IF STATE = BYTE#1 AND NOT FIFO.FULL THEN (* Anmelden *)
	(* nur eintragen wenn maximale anzahl nicht ueberschritten wurde *)
	tmp := BYTE_TO_INT(ID);
	IF FIFO.Y[tmp] < FIFO.MAX_ID THEN
		FIFO.Y[tmp] := USINT_TO_BYTE(BYTE_TO_USINT(FIFO.Y[tmp]) + USINT#1); (* IP_ID Zähler +1 *)
		tmp := FIFO.NW; (* geht bei mir leider nicht anders *)
		FIFO.X[tmp] := ID;
		IF FIFO.NW = FIFO.TOP THEN FIFO.NW := 1; ELSE FIFO.NW := FIFO.NW + 1; END_IF;
		FIFO.FULL := FIFO.NW = FIFO.NR;
		FIFO.EMPTY := FALSE;
		STATE := BYTE#2; (* weiterschalten auf "Warten auf Freigabe" *)
		(*####################  DEBUG-MESSAGE  ###################################*)
		(*IF _debug_enable THEN
			LOG_CL.NEW_MSG := 'FIFO: ADD ID:~1';
			LOG_CL.PRINTF[1]  := BYTE_TO_STRING(ID);
			LOG_MSG();
		END_IF;*)
		(*########################################################################*)

	END_IF;
END_IF;

IF STATE = BYTE#2 AND NOT FIFO.EMPTY THEN (* check current stack element *)
	tmp := FIFO.NR; (* geht bei mir leider nicht anders *)
	IF ID = FIFO.X[tmp] THEN
	STATE := BYTE#3; (* weiterschalten auf "Zugriffsfreigabe" *)
	END_IF;
END_IF;

IF STATE = BYTE#4 AND NOT FIFO.EMPTY THEN (* remove from stack *)
	tmp := FIFO.NR; (* geht bei mir leider nicht anders *)
	IF ID = FIFO.X[tmp] THEN
		tmp := BYTE_TO_INT(ID); (* geht bei mir leider nicht anders *)
		FIFO.Y[tmp] := USINT_TO_BYTE(BYTE_TO_USINT(FIFO.Y[tmp]) - USINT#1); (* ID Zähler -1 *)
		IF FIFO.NR = FIFO.TOP THEN FIFO.NR := 1; ELSE FIFO.NR := FIFO.NR + 1; END_IF;
		FIFO.EMPTY := FIFO.NR = FIFO.NW;
		FIFO.FULL := FALSE;
		(*####################  DEBUG-MESSAGE  ###################################*)
		(*IF _debug_enable THEN
			LOG_CL.NEW_MSG := 'FIFO: REMOVE ID:~1';
			LOG_CL.PRINTF[1]  := BYTE_TO_STRING(ID);
			LOG_MSG();
		END_IF;*)
		(*########################################################################*)
	END_IF;
	STATE := BYTE#5; (* "Remove done" *)
END_IF;

(* revision history
ks	18. oct. 2008	rev 1.0
	original version

*)

END_FUNCTION_BLOCK

// oscat_network/POUs/OTHER/ELEMENT_GET
FUNCTION ELEMENT_GET : STRING(ELEMENT_LENGTH)
VAR_INPUT
	SEP : BYTE;
	POS : INT;
END_VAR
VAR_IN_OUT
	ELEMENT : STRING(ELEMENT_LENGTH);
END_VAR
VAR
	i : INT := 1;
	o : INT := 1;
	pt : POINTER TO ARRAY[1..ELEMENT_LENGTH] OF BYTE;
	po : POINTER TO ARRAY[1..ELEMENT_LENGTH] OF BYTE;
	cnt: INT;
	c: BYTE;
END_VAR

(*
version 1.0	05. apr. 2011
programmer 	ks
tested by		kst

ELEMENT_GET liefert das element an der stelle pos einer liste.
die liste liegt als string von elementen vor die mit den zeichen SEP separiert sind.

*)

(* load pointers *)
pt := ADR(ELEMENT);
po := ADR(ELEMENT_GET);

(* search for the n-th occurence of a separation character and store position in i *)
WHILE (cnt < pos) AND (i < ELEMENT_LENGTH) AND (pt^[i] > 0) DO
	IF pt^[i] = sep THEN cnt := cnt + 1; END_IF;
	i := i + 1;
END_WHILE;

(* copy the list element to output *)
IF i < ELEMENT_LENGTH THEN c := pt^[i]; END_IF;
WHILE (c <> sep) AND (c > 0) AND (o < ELEMENT_LENGTH) AND (i < ELEMENT_LENGTH) DO
	po^[o] :=pt^[i];
	o := o + 1;
	i := i + 1;
	c := pt^[i];
END_WHILE;

(* terminate the output string *)
po^[o] := 0;

(* revision histroy
ks 05. apr. 2011	rev 1.0
	original release

*)

END_FUNCTION

// oscat_network/POUs/OTHER/ELEMENT_COUNT
FUNCTION ELEMENT_COUNT : INT
VAR_INPUT
	SEP : BYTE;
END_VAR
VAR_IN_OUT
	ELEMENT : STRING(ELEMENT_LENGTH);
END_VAR
VAR
	pt : POINTER TO ARRAY[1..ELEMENT_LENGTH] OF BYTE;
	l: INT;
	pos: INT;
END_VAR

(*
version 1.0	05. apr. 2011
programmer 	hugo
tested by		oscat

ELEMENT_COUNT liefert die anzahl der elemente einer liste.
die liste liegt als string von elementen vor die mit den zeichen SEP separiert sind.

*)

IF ELEMENT = '' THEN
	ELEMENT_COUNT := 0;
ELSE
	PT := ADR(ELEMENT);
	ELEMENT_COUNT := 1;
	l := LEN(ELEMENT);
	FOR pos := 1 TO l DO
		IF pt^[pos] = SEP THEN ELEMENT_COUNT := ELEMENT_COUNT + 1; END_IF;
	END_FOR;
END_IF;

(* revision histroy
ks	5. apr. 2011	rev 1.0
	original release

*)

END_FUNCTION

// oscat_network/POUs/DATA_LOG/DLOG_FILE_TO_SMTP_1
(* @OBJECTFLAGS := '0, 8' *)
FUNCTION_BLOCK DLOG_FILE_TO_SMTP_1
VAR_IN_OUT
	SERVER : STRING;
	MAILFROM : STRING;
	MAILTO : STRING(STRING_LENGTH);
	SUBJECT : STRING;
	BODY : STRING(STRING_LENGTH);
	X : DLOG_DATA;
END_VAR
VAR_INPUT
	FILE_DELETE : BOOL;
	TIMEOUT : TIME := T#30s;
	DTI : DT;
	DTI_OFFSET : INT;
	RETRY : INT;
	RETRY_TIME : TIME := T#30s;
	DNS_IP4 : DWORD;
END_VAR
VAR_OUTPUT
	DONE : BOOL;
	BUSY : BOOL;
	ERROR_C : DWORD;
	ERROR_T : BYTE;
END_VAR
VAR
	UCBD : UNI_CIRCULAR_BUFFER_DATA;
	UCB : UNI_CIRCULAR_BUFFER;
	SMTP_CLIENT : SMTP_CLIENT;
	WT_1 : TON;
	ftrig_old : BOOL;
	files : STRING(STRING_LENGTH);
	step : INT;
	smtp_busy : BOOL;
	smtp_done : BOOL;
	cnt : INT;

	(*LOG_MSG : LOG_MSG;
	_debug_enable : BOOL := TRUE;*)
END_VAR

(*
version 1.2		26. july. 2011
programmer		ks
tested by			ks

DLOG_FILE_TO_SMTP der Baustein versendet die vom DLOG_STORE_FILE_CSV erzeugten Dateien als Email
*)

(* neue Filenamen speichern *)
IF X.NEW_FILE_RTRIG AND ftrig_old = FALSE THEN
	UCBD.D_HEAD := 1;
	UCBD.D_MODE := 1;
	UCBD.D_STRING := X.NEW_FILE;
	UCB(DATA:=UCBD); (* Daten eintragen *)
END_IF;
ftrig_old := X.NEW_FILE_RTRIG;

CASE step OF

00:	IF UCBD.BUF_COUNT > 0 AND smtp_busy = FALSE THEN
		UCBD.D_MODE := 12; (* Daten lesen und löschen *)
		UCB(DATA:=UCBD);
		files := UCBD.D_STRING;
		IF FILE_DELETE THEN
			files := CONCAT(files,';#DEL#');
		END_IF;
		cnt := 0;
		step := 10;
	END_IF;

10:	IF smtp_busy = FALSE THEN
		IF smtp_done THEN
			(*####################  DEBUG-MESSAGE  ###################################*)
			(*IF _debug_enable THEN
				LOG_CL.NEW_MSG := 'F_T_SMTP: /FILE OK >~1<';
				LOG_CL.PRINTF[1] := files;
				LOG_MSG();
			END_IF;*)
			(*########################################################################*)
			step := 0;
		ELSE
			step := 20; (* pause nach error *)
		END_IF;
	END_IF;

20:	IF WT_1.Q THEN (* Wartezeit *)
		cnt := cnt - 1;
		IF RETRY = 0 THEN (* Transfer unbegrenzt wiederholen *)
			(*####################  DEBUG-MESSAGE  ###################################*)
			(*IF _debug_enable THEN
				LOG_CL.NEW_MSG := 'F_T_SMTP: Auftrag unbegrenzt wiederholen /file: ~2';
				LOG_CL.PRINTF[2] := files;
				LOG_MSG();
			END_IF;*)
			(*########################################################################*)
			step := 10; (* Transfer wiederholen *)
		ELSIF cnt >= 0 THEN
			(*####################  DEBUG-MESSAGE  ###################################*)
			(*IF _debug_enable THEN
				LOG_CL.NEW_MSG := 'F_T_SMTP: Auftrag wiederholen /cnt: ~1 /file: ~2';
				LOG_CL.PRINTF[1] := INT_TO_STRING(cnt);
				LOG_CL.PRINTF[2] := files;
				LOG_MSG();
			END_IF;*)
			(*########################################################################*)
			step := 10; (* Transfer wiederholen *)
		ELSE
			(*####################  DEBUG-MESSAGE  ###################################*)
			(*IF _debug_enable THEN
				LOG_CL.NEW_MSG := 'F_T_SMTP: Auftrag verworfen /file: ~2';
				LOG_CL.PRINTF[2] := files;
				LOG_MSG();
			END_IF;*)
			(*########################################################################*)
			step := 0; (* Auftrag verwerfen *)
		END_IF;
	END_IF;

END_CASE;

BUSY := step = 10;
DONE := step = 0;
WT_1(IN:= step = 20, PT:= RETRY_TIME);

SMTP_CLIENT(
	ACTIVATE:= BUSY,
	TIMEOUT:= TIMEOUT,
	DTI:= DTI,
	DTI_OFFSET:= DTI_OFFSET,
	DNS_IP4:= DNS_IP4,
	SERVER:= SERVER,
	MAILFROM:= MAILFROM,
	MAILTO:= MAILTO,
	SUBJECT:= SUBJECT,
	BODY:= BODY,
	FILES:= FILES,
	DONE=> smtp_done,
	BUSY=> smtp_busy,
	ERROR_C=> ERROR_C,
	ERROR_T=> ERROR_T
	);

(* revision history

ks	01. jan. 2011	rev 1.0
	original version

ks	28. apr. 2011	rev 1.1
	stringfehler bei option 'file_delete'

ks	26. july. 2011	rev 1.2
	Codeoptimierung D_MODE 12
*)

END_FUNCTION_BLOCK

// oscat_network/POUs/NETWORK/SMTP_CLIENT
FUNCTION_BLOCK SMTP_CLIENT
VAR_INPUT
	ACTIVATE : BOOL;
	TIMEOUT : TIME;
	DTI : DT;
	DTI_OFFSET : INT;
	DNS_IP4 : DWORD;
END_VAR
VAR_OUTPUT
	DONE : BOOL;
	BUSY : BOOL;
	ERROR_C : DWORD;
	ERROR_T : BYTE;
END_VAR
VAR_IN_OUT
	SERVER : STRING;
	MAILFROM : STRING;
	MAILTO : STRING(STRING_LENGTH);
	SUBJECT : STRING;
	BODY : STRING(STRING_LENGTH);
	FILES : STRING(STRING_LENGTH);
END_VAR
VAR
	IP_C : IP_C; (* IP_Control Verwaltungsstruktur *)
	S_BUF : NETWORK_BUFFER;
	R_BUF : NETWORK_BUFFER;
	F_BUF : NETWORK_BUFFER;
	URL_DATA : url;
	DNS_CLIENT : DNS_CLIENT;
	IPC : IP_CONTROL;
	FS : FILE_SERVER;
	FSD : FILE_SERVER_DATA;
	BASE64_ENCODE_STR : BASE64_ENCODE_STR;
	BASE64_ENCODE_STREAM : BASE64_ENCODE_STREAM;
	fpd : FILE_PATH_DATA;
	MD5_CRAM_AUTH : MD5_CRAM_AUTH;
	MD5_RUN : BOOL;
	activate_last : BOOL;
	step : INT;
	snd_step : INT;
	str1 : STRING(STRING_LENGTH);
	str2 : STRING(STRING_LENGTH);
	str3 : STRING;
	snd_text :	STRING(STRING_LENGTH);
	snd_lf_cnt : INT;
	rcv_text :	STRING(STRING_LENGTH);
	rcv_s : STRING(3);
	rcv_state : INT;
	auth_names : STRING := ' PLAIN; LOGIN; CRAM-MD5';
	auth_state : BYTE;
	TON_WAIT : TON;
	last_step : INT;
	next_step : INT;
	timeout2 : TIME;
	timeout3 : TIME;
	last_block : BOOL;
	file_delete : BOOL;
	esmtp : BOOL;
	cnt1 : INT;
	cnt2 : INT;
	cnt3 : INT;
	cnt4 : INT;
	idx1 : INT;
	idx2 : INT;
	idx3 : INT;
	snd_idx : INT;
	snd_enable : BOOL;
	i1 : INT;
	b64_done : BOOL;
	b64_start : BOOL;
	b64_max : UINT := 2880; (* short = 960 / long = 2880 *)
	b64_buf1 : ARRAY [0..47] OF BYTE;
	b64_buf2 : ARRAY [0..63] OF BYTE;
	b64_size1 : INT;
	b64_size2 : INT;
	b64_lf : BOOL;
	b64_str1	: STRING(144);
	b64_str2	: STRING(192);
	md5_user : STRING(64);
	md5_password : STRING(64);
	md5_b64_ts : STRING(64);
	md5_auth_key : STRING(192);
	ip_c_red_disable : BOOL; (* IP_CONTROL - Remote Disconnect Error unterdrücken *)

	(*LOG_MSG : LOG_MSG;
	_debug_enable : BOOL := TRUE;*)
END_VAR

(*
version 1.3		30. may 2011
programmer		ks
tested by			ks

SMTP_CLIENT versendet Email an verschiedene Emailadressen mit optionalen Dateianhängen.



mögliche Rückgabecodes:

Grad der Schwere
 
Die erste Stelle des Rückgabecodes gibt den Grad der Schwere an:
1yz Vorläufige positive Antwort
2yz Antwort über positiven Abschluss 
3yz Positive Zwischenantwort 
4yz Antwort über vorübergehenden negativen Abschluss 
5yz Permanente negative Antwort 
 
Die zweite Stelle gibt die Kategorie der Antwort an: 
x0z Syntaxfehler 
x1z Information 
x2z Verbindung 
x3z Nicht festgelegt 
x4z Nicht festgelegt 
x5z Mail-System 
 
Die dritte Stelle dient zur genaueren Bestimmung der Kategorie. 

Betriebsprotokolle enthalten folgende Codes: 
211 	Systemstatus oder Hilfe-Antwort des Systems  
214 	Hilfe-Nachricht - Informationen zur Verwendung des Empfängers oder zur  
      	Bedeutung eines bestimmten nicht standardmäßigen Befehls; wobei  
      	diese Antwort nur für Personen hilfreich ist, nicht für Systeme 
220 	Service ready (Dienst bereit) 
221 	Service closing transmission channel (Dienst schließt Übertragungskanal) 
235  Authentication succeeded (Authentifizierung erfolgreich)
250 	Requested mail action okay, completed (angeforderte Mail-Maßnahme ok und abgeschlossen) 
251 	User not local; will forward to (Benutzer nicht lokal; Weiterleitung an) 
252 	Cannot VRFY user, but will accept message and attempt delivery (kann Benutzer nicht überprüfen, aber akzeptiert Nachricht und versucht Auslieferung) 
354 	Start mail input; end with. (Mail-Eingabe starten; Ende mit .) 
421 	Service not available, closing transmission channel 	(Dienst nicht verfügbar, Übertragungskanal wird geschlossen) diese Antwort kann auf jeden Befehl folgen, wenn der Dienst weiß, dass er beendet werden muss 
450 	Requested mail action not taken: mailbox unavailable (angeforderte E-Mail-Maßnahme nicht ausgeführt, Mailbox nicht  verfügbar) - z. B. weil Mailbox besetzt 
451	 Requested action aborted: local error in processing (angeforderte Maßnahme abgebrochen: lokaler Fehler bei der Verarbeitung) 
452 	Requested action not taken: insufficient system storage (angeforderte Maßnahme abgebrochen: Systemspeicher nicht ausreichend) 
500 	Syntax error, command unrecognized (Syntaxfehler, Befehl nicht erkannt) - z. B. weil Befehlszeile zu lang 
501 	Syntax error in parameters or arguments (Syntaxfehler in Parametern oder Argumenten) 
502 	Command not implemented (Befehl nicht implementiert) 
504 	Command parameter not implemented (Befehlsparameter nicht implementiert) 
550 	Requested action not taken: mailbox unavailable (Angeforderte Maßnahme nicht ausgeführt: Mailbox nicht verfügbar) 
551 	User not local; please try (Benutzer nicht lokal; versuchen Sie es mit) 
552 	Requested mail action aborted: exceeded storage allocation (angeforderte Mail-Maßnahme abgebrochen: Speicherplatzzuweisung überschritten) 
553 	Requested action not taken: mailbox name not allowed (angeforderte Maßnahme nicht ausgeführt: Mailboxname nicht zulässig) 
554 	Transaction failed (Transaktion fehlgeschlagen) 

#########################
ERROR_T

1 = DNS_CLIENT
2 = SMTP Steuerkanal
4 = FILE_SERVER
5 = Ablaufstörung
#########################

*)

CASE step OF

00:	IF ACTIVATE AND NOT activate_last THEN
		TIMEOUT := MAX(T#10s,TIMEOUT);
		timeout2 := TIMEOUT + T#1s;
		timeout3 := TIMEOUT / 2;
		DONE := FALSE;
		ip_c_red_disable := FALSE;
		ERROR_C := DWORD#0;
		ERROR_T := BYTE#0;
		FSD.ERROR := BYTE#0;
		file_delete := FALSE;
		URL_DATA := STRING_TO_URL(STR:=SERVER,DEFAULT_PROTOCOL:='',DEFAULT_PATH:='/');
		idx1 := FIND(URL_DATA.USER,'%'); (* % Zeichen auf @ ändern *)
		IF idx1 > 0 THEN
			URL_DATA.USER := REPLACE(URL_DATA.USER,'@',1,idx1);
		END_IF;
		esmtp := LEN(URL_DATA.PASSWORD) > 0; (* SMTP oder ExtendedSMTP *)
		step := 10;
	END_IF;

10:	IF DNS_CLIENT.DONE THEN
		step := 20;
	ELSIF DNS_CLIENT.ERROR <> DWORD#0 THEN
		ERROR_C := DNS_CLIENT.ERROR;
		ERROR_T := BYTE#1;
		step := 980;
	END_IF;

20:	(* SMTP Kommunikation einrichten *)
	IP_C.C_PORT := SEL(URL_DATA.PORT = WORD#0,URL_DATA.PORT,WORD#25); (* Portnummer eintragen *)
  	IP_C.C_IP := DNS_CLIENT.IP4; (* IP eintragen *)
  	IP_C.C_MODE := BYTE#0; (* Mode: TCP+ACTIV+PORT *)
  	IP_C.TIME_RESET := TRUE; (* Zeitueberwachung rücksetzen *)
  	IP_C.C_ENABLE := TRUE; (* Verbindungsaufbau freigeben *)
  	IP_C.R_OBSERVE := TRUE; (* Empfangsueberwachung *)
	R_BUF.SIZE := UINT#0;
	snd_enable := TRUE; (* sofortiges senden erlauben *)
	snd_idx := 0;
	step := 30;

30:	IF rcv_state = 220 THEN (* 220 = Service ready *)
		IF esmtp THEN
			snd_text := 'EHLO OSCAT'; (* ExtendedSMTP *)
			next_step := 40;
		ELSE
			snd_text := 'HELO OSCAT'; (* SMTP *)
			next_step := 90;
		END_IF;
		snd_lf_cnt := 1;
	END_IF;

40:	IF rcv_state = 250 THEN (* 250 = Requested mail action okay, completed  *)
		auth_state := BYTE#0;
		str1 := auth_names;
		idx1 := 0;
		idx2 := 1900;
		step := 50;
	END_IF;

50:	str2 := ELEMENT_GET(59, idx1, str1); (* Trennzeichen >;< *)
	IF LEN(str2) > 0 THEN
		IF FIND(rcv_text,str2) > 0 THEN
			auth_state := BIT_LOAD_B(auth_state, TRUE, idx1);
			str3 := str2; (* aktuellen AUTH-Type Namen sichern *)
			idx2 := 1000 + (idx1 * 100); (* Schritt berechnen *)
		END_IF;
		idx1 := idx1 + 1;
	ELSE
		step := 60;
	END_IF;

60:	IF rcv_state = 250 THEN (* 250 = Requested mail action okay, completed  *)
		snd_text := CONCAT('AUTH',str3);
		next_step := idx2; (* mit den jeweiligen Authentifizierung Schritten fortfahren *)
	END_IF;

 (* ++++++++++++++++++++++++++++++++++++++++++++++++++++++*)

90:	IF rcv_state = 235 OR rcv_state = 250 THEN (* 235 = Authentication successful / 250 Requested mail action okay *)
		str2 := MAILFROM;
		str1 := ELEMENT_GET(59, 1, str2);(* Angezeigter Name lesen , Trennzeichen >;< *)
		IF LEN(str1) > 0 THEN
			str3 := INSERT('"" ', str1, 1);
		ELSE
			str3 := '';
		END_IF;
		str1 := ELEMENT_GET(59, 0, str2);(* MAILFROM lesen , Trennzeichen >;< *)
		str2 := INSERT('MAIL FROM: <>', str1, 12);
		snd_text := INSERT(str2, str3, 11);
		str3 := snd_text; (* zur wiederverwendung speichern *)
		next_step := 95;
		cnt1 := ELEMENT_COUNT(35, MAILTO); (* Trennzeichen >#< , Anzahl der Blöcke bestimmen *)
		cnt2 := 0;
	END_IF;

95:	IF rcv_state = 250 THEN (* 250 = Requested mail action okay *)
		IF cnt2 < cnt1 THEN
			str1 := ELEMENT_GET(35, cnt2, MAILTO);(* Trennzeichen >#< *)
			cnt3 := ELEMENT_COUNT(59, str1); (* Trennzeichen >;< , Anzahl der Sub-Blöcke bestimmen *)
			cnt4 := 0;
			cnt2 := cnt2 + 1;
			step := 100; (* Blockinhalt auswerten *)
		ELSE
			step := 110; (* alle Blöcke bearbeitet *)
		END_IF;
	END_IF;

100:	IF rcv_state = 250 THEN (* 250 = Requested mail action okay *)
		IF cnt4 < cnt3 THEN
			str2 := ELEMENT_GET(59, cnt4, str1); (* Trennzeichen >;< *)
			snd_text := INSERT('RCPT TO: <>', str2, 10);
			cnt4 := cnt4 + 1;
			next_step := 100;
		ELSE
			step := 95;
		END_IF;
	END_IF;

110:	IF rcv_state = 250 THEN (* 250 = Requested mail action okay *)
		snd_text := 'DATA';
		next_step := 120;
	END_IF;

120:	IF rcv_state = 354 THEN (* 354 = Start mail input; end with. *)
		snd_enable := FALSE;
		snd_text := REPLACE(str3, 'From', 9, 1); (* 'MAIL FROM' durch "From" ersetzen *)
		cnt2 := 0;
		cnt1 := MIN(2,cnt1); (* BlindCopy Block ausblenden *)
		step := 200;
	END_IF;

200:	IF snd_step = 0 THEN
		IF cnt2 < cnt1 THEN
			str1 := ELEMENT_GET(35, cnt2, MAILTO);(* Trennzeichen >#< *)
			cnt3 := ELEMENT_COUNT(59, str1); (* Trennzeichen >;< , Anzahl der Sub-Blöcke bestimmen *)
			cnt4 := 0;
			cnt2 := cnt2 + 1;
			str3 := SEL(cnt2 = 1,'Cc: <>','To: <>');
			step := 205; (* Blockinhalt auswerten *)
		ELSE
			step := 210; (* alle Blöcke bearbeitet *)
		END_IF;
	END_IF;

205:	IF snd_step = 0 THEN
		IF cnt4 < cnt3 THEN
			str2 := ELEMENT_GET(59, cnt4, str1); (* Trennzeichen >;< *)
			snd_text := INSERT(str3, str2, 5);
			cnt4 := cnt4 + 1;
		ELSE
			step := 200;
		END_IF;
	END_IF;

210:	IF snd_step = 0 THEN
		snd_text := CONCAT('Subject: ',SUBJECT);
		step := 220;
	END_IF;

220:	IF snd_step = 0 THEN
		DTI := UDINT_TO_DT(DT_TO_UDINT(DTI) + INT_TO_UDINT(- DTI_OFFSET * 60)); (* Minuten-Offset auf Sekunden umrechnen und addieren *)
		IF esmtp THEN (* ESMTP Format >Date: Thu, 21 May 1998 05:33:29 -0700< *)
			str2 := ';Mon;Tue;Wed;Thu;Fri;Sat;Sun';
			str1 := ELEMENT_GET(59, DAY_OF_WEEK(DT_TO_DATE(DTI)), str2);
			snd_text := CONCAT('Date: ',str1);
			str1 := DT_TO_STRF(DTI, 0, ', #H #E #A #N:#R:#T +0000', 1);
			snd_text := CONCAT(snd_text,str1);
		ELSE (* SMTP Format >Date: 21 May 98 05:33:29< *)
			snd_text := DT_TO_STRF(DTI, 0, 'Date: #G #E #B #N:#R:#T', 1);
		END_IF;
		step := 230;
	END_IF;

230:	IF snd_step = 0 THEN
		snd_text := 'MIME-Version: 1.0';
		step := 250;
	END_IF;

250:	IF snd_step = 0 THEN
		snd_text := 'Content-Type: multipart/mixed;boundary="x"';
		snd_lf_cnt := 2;
		step := 260;
	END_IF;

260:	IF snd_step = 0 THEN
		snd_enable := TRUE;
		snd_text := 'This is a multi-part message in MIME format.';
		step := 270;
	END_IF;

270:	IF snd_step = 0 THEN
		snd_enable := FALSE;
		snd_text := '--x';
		snd_lf_cnt := 1;
		step := 280;
	END_IF;

280:	IF snd_step = 0 THEN
		snd_text := 'Content-Type: text/plain; format=flowed; charset="iso-8859-1";';
		snd_text := CONCAT(snd_text,' reply-type=original'); (* PCWORX kann nur konstanten mit max 80 zeichen *)
		step := 290;
	END_IF;

290:	IF snd_step = 0 THEN
		snd_text := 'Content-Transfer-Encoding: 8bit';
		snd_lf_cnt := 2;
		step := 300;
	END_IF;

300:	IF snd_step = 0 THEN
		snd_enable := TRUE;
		snd_text := BODY;
		snd_lf_cnt := 2;
		step := 310;
	END_IF;

310:	IF snd_step = 0 THEN
		cnt1 := ELEMENT_COUNT(59, FILES) - 1; (* Anzahl der Dateien *)
		step := 400;
	END_IF;

(* +++++++++++++ File-Attachment ++++++++++++ *)
400:	IF cnt1 >= 0 THEN
		str1 := ELEMENT_GET(59, cnt1, FILES);
		FILE_PATH_SPLIT(FILENAME:=str1,X:=fpd); (* Datei-Path zerlegen *)
		IF fpd.FILENAME = '#DEL#' THEN
			file_delete := TRUE;
		ELSE
			step := 410;
		END_IF;
		cnt1 := cnt1 - 1;
	ELSE
		step := 800;
	END_IF;

410:	IF snd_step = 0 THEN
		snd_enable := FALSE;
		snd_text := '--x';
		snd_lf_cnt := 1;
		step := 420;
	END_IF;

420:	IF snd_step = 0 THEN
		snd_text := 'Content-Transfer-Encoding: BASE64';
		str2 := CONCAT(fpd.FILENAME,'"');
		step := 430;
	END_IF;

430:	IF snd_step = 0 THEN
		snd_text := CONCAT('Content-Type: application/octet-stream; name="',str2);
		step := 440;
	END_IF;

440:	IF snd_step = 0 THEN
		snd_enable := TRUE;
		snd_text := CONCAT('Content-Disposition: attachment; filename="',str2);
		snd_lf_cnt := 2;
		step := 450;
	END_IF;

450:	IF snd_step = 0 THEN
		FSD.FILENAME := str1; (* Dateiname *)
		FSD.OFFSET := UDINT#0; (* Start bei Dateianfang *)
		FSD.AUTO_CLOSE := T#0s; (* kein Auto-Close verwenden *)
		step := 460;
	END_IF;

460:	FSD.MODE := BYTE#1; (* vorhandene Datei zum lesen öffnen *)
	F_BUF.SIZE := b64_max; (* maximale länge einlesen *)
	idx1 := 0;
	idx2 := 0;
	step := 470;

470:	IF FSD.MODE = BYTE#0 AND FSD.ERROR = BYTE#0 THEN
		last_block := FSD.FILE_SIZE = FSD.OFFSET;
		b64_size1 := MIN(48,UINT_TO_INT(F_BUF.SIZE) - idx1);
		IF b64_size1 > 0 THEN
			idx3 := b64_size1 - 1;
			FOR i1 := 0 TO idx3 DO (* daten in BASE64 buffer kopieren *)
				b64_buf1[i1] := F_BUF.BUFFER[idx1];
				idx1 := idx1 + 1;
			END_FOR;
			BASE64_ENCODE_STREAM( SIZE1:= b64_size1, BUF1:= b64_buf1, BUF2:= b64_buf2, SIZE2=> b64_size2); (* BASE64 Kodierung *)
			idx3 := b64_size2 - 1;
			FOR i1 := 0 TO idx3 DO (* Daten aus BASE64 buffer kopieren *)
				S_BUF.BUFFER[idx2] := b64_buf2[i1];
				idx2 := idx2 + 1;
			END_FOR;
			b64_lf := TRUE;
			(*####################  DEBUG-MESSAGE  ###################################*)
			(*IF _debug_enable THEN
				LOG_CL.NEW_MSG := 'B64: FILE ~1 /SIZE ~2 /OFF ~3 /BSIZE ~4 /idx1 ~5 /idx2 ~6';
				LOG_CL.PRINTF[1] := FSD.FILENAME;
				LOG_CL.PRINTF[2] := UDINT_TO_STRING(FSD.FILE_SIZE);
				LOG_CL.PRINTF[3] := UDINT_TO_STRING(FSD.OFFSET);
				LOG_CL.PRINTF[4] := INT_TO_STRING(b64_size1);
				LOG_CL.PRINTF[5] := INT_TO_STRING(idx1);
				LOG_CL.PRINTF[6] := INT_TO_STRING(idx2);
				LOG_MSG();
			END_IF;*)
			(*########################################################################*)
		ELSE
			b64_lf := last_block;
			step := 480; (* block beendet  *)
		END_IF;
		IF b64_lf THEN
			S_BUF.BUFFER[idx2] := BYTE#16#0D;
			idx2 := idx2 + 1;
			S_BUF.BUFFER[idx2] := BYTE#16#0A;
			idx2 := idx2 + 1;
		END_IF;
		(*####################  DEBUG-MESSAGE  ###################################*)
		(*IF _debug_enable THEN
			LOG_CL.NEW_MSG := 'B64: exit ~1 /SIZE ~2 /OFF ~3 /eof ~4 /lf_cnt ~5';
			LOG_CL.PRINTF[1] := FSD.FILENAME;
			LOG_CL.PRINTF[2] := UDINT_TO_STRING(FSD.FILE_SIZE);
			LOG_CL.PRINTF[3] := UDINT_TO_STRING(FSD.OFFSET);
			LOG_CL.PRINTF[4] := BOOL_TO_STRING(last_block);
			LOG_CL.PRINTF[5] := INT_TO_STRING(snd_lf_cnt);
			LOG_MSG();
		END_IF;*)
		(*########################################################################*)
	END_IF;

480:	S_BUF.SIZE := INT_TO_UINT(idx2); (* Daten senden *)
	(*####################  DEBUG-MESSAGE  ###################################*)
	(*IF _debug_enable THEN
		LOG_CL.NEW_MSG := 'B64: tcp_send ~1';
		LOG_CL.PRINTF[1] := INT_TO_STRING(idx2);
		LOG_MSG();
	END_IF;*)
	(*########################################################################*)
	step := 490;

490:	IF S_BUF.SIZE = UINT#0 THEN (* warten bis alle daten gesendet sind *)
		step := SEL(last_block ,460,400);
	END_IF;

(* ++++++++++++++++++++++++++++++++++++++++ *)

800:	IF snd_step = 0 THEN
		snd_enable := FALSE;
		snd_text := '--x--';
		snd_lf_cnt := 2;
		step := 810;
	END_IF;

810:	IF snd_step = 0 THEN
		snd_enable := TRUE;
		snd_text := '.';
		snd_lf_cnt := 1;
		step := 820;
	END_IF;

820:	IF rcv_state = 250 THEN (* 250 = Requested mail action okay *)
		snd_text := 'QUIT';
		ip_c_red_disable := TRUE;
		next_step := 830;
	END_IF;

830:	IF rcv_state = 221  OR TON_WAIT.ET > timeout3 THEN (* 221 = Service closing transmission channel *)
		step := 900;
	END_IF;

(* ================================================== *)

900:IF FILE_DELETE THEN (* Dateien nach transfer löschen *)
		cnt1 := ELEMENT_COUNT(59, FILES) - 1; (* Anzahl der Dateien *)
		step := 910;
	ELSE
		step := 950;
	END_IF;

910:	IF FSD.MODE = BYTE#0 AND FSD.ERROR = BYTE#0 THEN
		IF cnt1 >= 0 THEN
			str1 := ELEMENT_GET(59, cnt1, FILES);
			IF str1 <> '#DEL#' THEN
				FSD.FILENAME := str1;
				FSD.MODE := BYTE#4; (* File Remove *)
			END_IF;
			cnt1 := cnt1 - 1;
		ELSE
			step := 950;
		END_IF;
	END_IF;

950:DONE := TRUE;
	step := 980;

980:IP_C.C_ENABLE := FALSE; (* SMTP Steuerkanal schliessen *)
	S_BUF.SIZE := UINT#0;
	R_BUF.SIZE := UINT#0;
	snd_step := 0;
	next_step := 0;
	FSD.MODE := BYTE#5; (* Datei schliessen *)
	step := 990;

990:IF IP_C.C_STATE = BYTE#0 AND FSD.FILE_OPEN = FALSE THEN
		step := 0;
	END_IF;

(*  +++++++++++++++++ Authentifizierung +++++++++++++++++ *)

(* PLAIN ++++++++++++++++++++++++++++++++++++++++++++++++++++++++++ *)
1000:IF rcv_state = 334 THEN (* 334 = Authentifizierung  *)
		cnt1 := LEN(URL_DATA.USER);
		cnt2 := LEN(URL_DATA.PASSWORD);
		IF cnt1 + cnt2 <= 46 THEN (* USER + PASSWORD dürfen zusammen maximal 46 Zeichen haben *)
			b64_buf1[0] := BYTE#0;
			FOR i1 := 1 TO cnt1 DO
				b64_buf1[i1] := CODE(URL_DATA.USER, i1);
			END_FOR;
			b64_size1 := cnt1 + 1;
			b64_buf1[b64_size1] := BYTE#0;
			b64_size1 := b64_size1 + 1;
			FOR i1 := 1 TO cnt2 DO
				b64_buf1[b64_size1] := CODE(URL_DATA.PASSWORD, i1);
				b64_size1 := b64_size1 + 1;
			END_FOR;
			BASE64_ENCODE_STREAM( SIZE1:= b64_size1, BUF1:= b64_buf1, BUF2:= b64_buf2, SIZE2=> b64_size2); (* BASE64 Kodierung *)
			idx1 := b64_size2 - 1;
			FOR i1 := 0 TO idx1 DO
				S_BUF.BUFFER[i1] := b64_buf2[i1];
			END_FOR;
			S_BUF.BUFFER[b64_size2] := BYTE#16#0D;
			b64_size2 := b64_size2 + 1;
			S_BUF.BUFFER[b64_size2] := BYTE#16#0A;
			b64_size2 := b64_size2 + 1;
			S_BUF.SIZE := INT_TO_UINT(b64_size2);
			rcv_state := 0;
		END_IF;
		step := 90;
	END_IF;

(* LOGIN ++++++++++++++++++++++++++++++++++++++++++++++++++++++++++ *)
1100:IF rcv_state = 334 THEN (* 334 = Authentifizierung  *)
		b64_str1 := URL_DATA.USER;
		b64_start := TRUE; (* BASE64 kodierung von Username *)
		step := 1120;
	END_IF;

1120:IF b64_start AND b64_done THEN
		b64_start := FALSE;
		snd_text := b64_str2;
		next_step := 1130;
	END_IF;

1130:IF rcv_state = 334 THEN (* 334 = Password:  *)
		b64_str1 := URL_DATA.PASSWORD;
		b64_start := TRUE; (* BASE64 kodierung von Password *)
		step := 1140;
	END_IF;

1140:IF b64_start AND b64_done THEN
		b64_start := FALSE;
		snd_text := b64_str2;
		next_step := 90;
	END_IF;

(* CRAM-MD5 (Challenge-Response Authentication Mechanism, Message Digest 5) Authentifizierung auf Basis von MD5-HMAC-Algorithmus. *)
1200:IF rcv_state = 334 THEN (* 334 = Authentifizierung  *)
		md5_b64_ts := RIGHT(rcv_text,LEN(rcv_text) - 4);
		md5_user := URL_DATA.USER;
		md5_password := URL_DATA.PASSWORD;
		MD5_RUN := TRUE;
		step := 1220;
	END_IF;

1220:MD5_CRAM_AUTH(RUN:=MD5_RUN,USERNAME:=md5_user,PASSWORD:=md5_password,B64_TS:=md5_b64_ts,AUTH_KEY:=md5_auth_key);
	IF NOT MD5_RUN THEN
		snd_text := md5_auth_key;
		step := 90;
	END_IF;

(* keine Authentifizierung gefunden +++++++++++++++++++++++++++++++ *)
1900: ; (* Auf Laufzeitfehler warten *)

END_CASE;
(* ++++++++++++++++++++++++++++++++++++++++++++++++++++++++++ *)
IF step >= 30 THEN
	IF R_BUF.SIZE > UINT#0 THEN (* Daten wurden empfangen ? *)
		idx1 := UINT_TO_INT(R_BUF.SIZE);
		REPEAT (* zeilenterminierung erkennen und echtes TEXT-Ende bestimmen *)
			idx1 := idx1 - 1;
		UNTIL idx1 = 0 OR R_BUF.BUFFER[idx1] >= BYTE#32 (* TRUE = EXIT *)
		END_REPEAT;
		FOR i1 := 0 TO idx1 DO (* bei multiline alle CRLF durch >^< ersetzen *)
			IF R_BUF.BUFFER[i1] < BYTE#32 THEN
				R_BUF.BUFFER[i1] := BYTE#94; (* >^< *)
			END_IF;
		END_FOR;
		rcv_text := BUFFER_TO_STRING(PT:=ADR(R_BUF.BUFFER),SIZE:=idx1+1,START:=0,STOP:=STRING_LENGTH-1);
		IF LEN(rcv_text) >= 3 THEN (* Statuscode prüfen und auswerten *)
			rcv_s := LEFT(rcv_text,3);
			IF IS_NUM(STR:=rcv_s) THEN (* enthält nur Zahlen ? *)
				rcv_state := STRING_TO_INT(rcv_s);
			END_IF;
			IP_C.R_OBSERVE := FALSE;
		END_IF;
		R_BUF.SIZE := UINT#0; (* daten löschen *)

		(*####################  DEBUG-MESSAGE  ###################################*)
		(*IF _debug_enable THEN
			LOG_CL.NEW_MSG := 'RCV: >~1<';
			LOG_CL.PRINTF[1] := rcv_text;
			LOG_MSG();
		END_IF;*)
		(*########################################################################*)

	END_IF;
END_IF;

(* automatisches Datensenden *)

CASE snd_step OF

00:	IF LEN(snd_text) > 0 THEN

		(*####################  DEBUG-MESSAGE  ###################################*)
		(*IF _debug_enable THEN
			LOG_CL.NEW_MSG := 'SND: >~1< /lf ~2';
			LOG_CL.PRINTF[1] := snd_text;
			LOG_CL.PRINTF[2] := INT_TO_STRING(snd_lf_cnt);
			LOG_MSG();
		END_IF;*)
		(*########################################################################*)

		_STRING_TO_BUFFER(str:=snd_text,pos:=snd_idx,pt:=ADR(S_BUF.BUFFER),size:=SIZEOF(S_BUF.BUFFER)); (* String in puffer kopieren *)
		snd_idx := snd_idx + LEN(snd_text);
		FOR i1 := 1 TO snd_lf_cnt DO
			S_BUF.BUFFER[snd_idx] := BYTE#16#0D;
			snd_idx := snd_idx + 1;
			S_BUF.BUFFER[snd_idx] := BYTE#16#0A;
			snd_idx := snd_idx + 1;
		END_FOR;
		snd_text := '';
		rcv_state := 9999; (* letzen SMTP Status löschen *)

		IF snd_enable THEN
			S_BUF.SIZE := INT_TO_UINT(snd_idx); (* Sendelänge eintragen *)
			R_BUF.SIZE := UINT#0; (* Empfangsbuffer rücksetzen *)
			IP_C.R_OBSERVE := step <= 120 OR step >= 820;
			snd_idx := 0;
			snd_step := 10;
		END_IF;
	END_IF;

10:	IF S_BUF.SIZE = UINT#0 THEN (* warten bis alle daten gesendet sind *)
		IF next_step <> 0 THEN
			step := next_step;
			next_step := 0;
		END_IF;
		snd_step := 0;
	END_IF;

END_CASE;

(* Globale Fehlerbehandlung für Haupt-Routine *)
IF ERROR_T = BYTE#0 AND step > 20 THEN (* noch kein Fehler gespeichert und Hauptroutine aktiv *)

	IF IP_C.ERROR > DWORD#0 AND IP_C.C_ENABLE AND NOT IP_C.TIME_RESET THEN  (* IP Control 1 *)
		IF ip_c_red_disable = FALSE OR IP_C.ERROR <> DWORD#16#FD000000 THEN
			ERROR_C := IP_C.ERROR;
			ERROR_T := BYTE#2;
			step := 980;
		END_IF;
	END_IF;

	IF FSD.MODE = BYTE#0 THEN
		IF FSD.ERROR > BYTE#0 THEN
			ERROR_C := BYTE_TO_DWORD(FSD.ERROR);
			ERROR_T := BYTE#4; (* Dateizugriff *)
			step := 980;
		END_IF;
	END_IF;
END_IF;

IF TON_WAIT.Q THEN (* Ablaufstörung - Schrittkette *)
	ERROR_C := SHL(INT_TO_DWORD(step),16) OR INT_TO_DWORD(rcv_state); (* aktuellen Schritt und letzten SMTP Status eintragen *)
	ERROR_T := BYTE#5;
	step := 980;
END_IF;

(* ######################################################## *)

DNS_CLIENT(IP_C:=IP_C, S_BUF:=S_BUF, R_BUF:=R_BUF, DOMAIN:=URL_DATA.DOMAIN, IP4_DNS:= DNS_IP4, ACTIVATE:=step=10); (* DNS-Client *)
IPC(IP:= DWORD#0, PORT:= WORD#0 , TIME_OUT:= TIMEOUT, IP_C:= IP_C, S_BUF:= S_BUF, R_BUF:= R_BUF); (* SMTP Steuerkanal *)
FS(FSD:=FSD,PT:=F_BUF); (* FILE_SERVER *)
BASE64_ENCODE_STR(RUN:= b64_start, STR1:= b64_str1, STR2:= b64_str2, DONE=> b64_done); (* BASE64 kodierung *)

TON_WAIT(IN:=step = last_step AND step > 0,PT:=timeout2);
last_step := step;
activate_last := ACTIVATE;
BUSY := step <> 0;

(* revision history
ks	01. jan. 2011	rev 1.0
	original version
ks	06. apr. 2011	rev 1.1
	list_len und list_get durch element_count und element_get ersetzt
ks	11. may 2011	rev 1.2
	ip_control - remote disconnect error ausblenden, und sonderbehandlung für pcworx
ks	30. may. 2011	rev 1.3
	fehler bei empfangsüberwachung
*)

END_FUNCTION_BLOCK

// oscat_network/POUs/DATA_LOG/DLOG_REAL_1
FUNCTION_BLOCK DLOG_REAL_1
VAR_IN_OUT
	X : DLOG_DATA;
END_VAR
VAR_INPUT
	VALUE : REAL;
	N : INT;
	D : STRING(1) := ',';
	COLUMN : STRING(40);
	DELTA : REAL;
END_VAR
VAR
	UCB : UNI_CIRCULAR_BUFFER;
	init : BOOL;
	id : WORD;
	delta_last : REAL;
	value_last : REAL;
END_VAR

(*
version 1.2		25. july. 2011
programmer		ks
tested by			ks

DLOG_REAL legt den REAL-Wert als STRING im FIFO-RING-Buffer ab um diesen mit den Baustein DLOG_STORE_*  aufzuzeichnen
*)

IF NOT init THEN
	init := TRUE;
	X.ID_MAX := X.ID_MAX + 1;
	id := WORD#16#0201; (* Quelltype REAL , Zieltype STRING *)
END_IF;

IF X.ADD_HEADER THEN
	X.UCB.D_STRING := COLUMN;
	X.UCB.D_HEAD := id;
	X.UCB.D_MODE := 1;
	UCB(DATA:=X.UCB); (* Daten eintragen *)
ELSIF X.ADD_DATA THEN
	X.UCB.D_STRING := REAL_TO_STRF(IN:=value_last,N:=N,D:=D);
	X.UCB.D_HEAD := id;
	X.UCB.D_MODE := 1;
	UCB(DATA:=X.UCB); (* Daten eintragen *)
	delta_last := value_last;
ELSIF DELTA <> 0.0 THEN
	IF VALUE <= (delta_last - DELTA) OR VALUE >= (delta_last + DELTA) THEN
		X.ADD_DATA_REQ := TRUE;
		delta_last := VALUE;
	END_IF;
END_IF;
value_last := VALUE;

(* revision history
ks	01. jan. 2011	rev 1.0
	original version

ks	17. may. 2011	rev 1.1
	DELTA Funktion integriert

ks	25. july.   2011	rev 1.2
	neue head information
*)

END_FUNCTION_BLOCK

// oscat_network/POUs/DATA_LOG/DLOG_STORE_FILE_CSV_1
FUNCTION_BLOCK DLOG_STORE_FILE_CSV_1
VAR_IN_OUT
	X : DLOG_DATA;
END_VAR
VAR_INPUT
	ENABLE : BOOL;
	TRIG_M : BOOL;
	TRIG_T : UDINT;
	FILENAME : STRING;
	DTI : DT;
	SEP : BYTE;
END_VAR
VAR_OUTPUT
	ERROR_C : DWORD;
	ERROR_T : BYTE;
END_VAR
VAR
	FS : FILE_SERVER;
	FSD : FILE_SERVER_DATA;
	PT : NETWORK_BUFFER;
	UCB : UNI_CIRCULAR_BUFFER;
	ra : BOOL;
	trig_m_last : BOOL;
	dti_last : DT := DT#2070-02-06-06:28:15;
	enable_last : BOOL;
	fn_last : STRING;
	fn : STRING;
	init : BOOL;
	step: INT;
	idx : INT;
	log_stop : BOOL;
	n : USINT;
END_VAR

(*
version 1.2		25. jul. 2011
programmer		ks
tested by			ks

DLOG_STORE_FILE_CSV der Baustein schreibt die DLOG Parameter in einen lokale Datei im CSV-Format
*)

X.DTI := DTI; (* Datum / Zeit eintragen *)
IF DTI <> dti_last THEN
	X.CLOCK_TRIG := TRUE;
	dti_last := DTI;
	X.STORE_TYPE := 2;
ELSE
	X.CLOCK_TRIG := FALSE;
END_IF;

IF X.ADD_HEADER = FALSE THEN (* wenn add-header und add-data gleichzeitig ansteht, dann add-data einen zyklus länger anstehen lassen *)
	X.ADD_DATA := FALSE;
END_IF;
X.ADD_HEADER := FALSE;

IF ENABLE THEN
	IF X.CLOCK_TRIG THEN
		fn := DT_TO_STRF(DTI, 0, FILENAME, 0); (* automatische Dateinamen generierung *)
		IF TRIG_T > 0 THEN (* automatischer Trigger *)
			ra := DT_TO_UDINT(DTI) MOD TRIG_T = 0;
		END_IF;
	ELSE
		ra := FALSE;
	END_IF;
	IF (TRIG_M AND NOT trig_m_last) OR ra OR X.ADD_DATA_REQ THEN (* manueller, automatischer oder externer Trigger *)
		X.ADD_DATA := TRUE; (* Daten loggen *)
	END_IF;
	IF NOT init THEN
		init := TRUE;
		X.ADD_HEADER := TRUE; (* Spaltenüberschriften übernehmen *)
	END_IF;
END_IF;
X.ADD_DATA_REQ := FALSE; (* externe Anforderung rücksetzen *)

IF (NOT ENABLE AND enable_last) OR (fn <> fn_last AND step > 0) THEN (* Neg. Flanke ENABLE - Log Stop *)
	fn_last := fn;
	X.UCB.D_HEAD := WORD#16#FF00;
	X.UCB.D_MODE := 1;
	UCB(DATA:=X.UCB); (* Element schreiben *)
	X.ADD_HEADER := TRUE; (* Spaltenüberschriften übernehmen *)
END_IF;

CASE step OF

00:	IF ENABLE THEN
		fn_last := fn;
		FSD.FILENAME := fn; (* Dateiname *)
		FSD.OFFSET := 0; (* Start bei Dateianfang *)
		FSD.AUTO_CLOSE := T#0s; (* Auto-Close *)
		step := 20;
	END_IF;

20:	IF X.UCB.BUF_COUNT > 0 THEN (* Einträge vorhanden *)
		X.UCB.D_MODE := 10;
		UCB(DATA:=X.UCB); (* Element lesen , aber noch nicht entfernen *)
		IF X.UCB.D_HEAD = WORD#16#FF00 THEN (* LOG_STOP Command *)
			X.UCB.D_MODE := 11;
			UCB(DATA:=X.UCB); (* Element entfernen *)
			log_stop := TRUE;
			step := 40; (* Daten schreiben *)
		ELSIF idx + LEN(X.UCB.D_STRING) + 2 < SIZEOF(PT) THEN (* Platz für Element vorhanden ? *)
			X.UCB.D_MODE := 11;
			UCB(DATA:=X.UCB); (* Element entfernen *)
			_STRING_TO_BUFFER(STR:=X.UCB.D_STRING, POS:=idx, PT:=ADR(PT.BUFFER), SIZE:=SIZEOF(PT.BUFFER));
			idx := idx + LEN(X.UCB.D_STRING);
			n := n + 1;
			IF n = X.ID_MAX THEN (* letztes Element einer Zeile *)
				n := USINT#0;
				PT.BUFFER[idx] := 16#0D;
				idx := idx + 1;
				PT.BUFFER[idx] := 16#0A;
			ELSE
				PT.BUFFER[idx] := SEP;
			END_IF;
			idx := idx + 1;
		ELSE
			step := 40; (* Daten schreiben *)
		END_IF;
	END_IF;

40:	IF idx > 0 THEN (* Daten schreiben *)
		FSD.MODE := 3; (* create + write *)
		PT.SIZE := idx; (* Datenlänge eintragen *)
		idx := 0;
	END_IF;
	step := 60;

60:	IF FSD.MODE = 0 THEN
		IF log_stop THEN
			log_stop := FALSE;
			FSD.MODE := 5; (* Datei schliessen *)
			X.NEW_FILE := FSD.FILENAME;
			X.NEW_FILE_RTRIG := FALSE;
			step := 80;
		ELSE
			step := 20;
		END_IF;
	END_IF;

80:	IF FSD.MODE = 0 THEN (* Datei schliessen beendet *)
		X.NEW_FILE_RTRIG := TRUE;
		step := 0;
	END_IF;

END_CASE;

trig_m_last := TRIG_M;
enable_last := ENABLE;
FS(FSD:=FSD,PT:=PT); (* FILE_SERVER *)

ERROR_C := FSD.ERROR;
ERROR_T := SEL(FSD.ERROR > 0,0,1);

(* revision history
ks	01. jan. 2011	rev 1.0
	original version

ks	13. may. 2011	rev 1.1
	ADD_DATA_REQ, ERROR_T, ERROR_C hinzugefügt

ks	25. july. 2011	rev 1.2
	HEAD Informationen geändert, neuer Spaltenzähler
*)

END_FUNCTION_BLOCK

// oscat_network/POUs/DATA_LOG/DLOG_STORE_FILE_HTML_1
FUNCTION_BLOCK DLOG_STORE_FILE_HTML_1
VAR_IN_OUT
	X : DLOG_DATA;
END_VAR
VAR_INPUT
	ENABLE : BOOL;
	TRIG_M : BOOL;
	TRIG_T : UDINT;
	FILENAME : STRING;
	DTI : DT;
	HTML_CAPTION : STRING;
	HTML_TABLE : STRING;
	HTML_TR_HEAD : STRING;
	HTML_TR_EVEN : STRING;
	HTML_TR_ODD : STRING;
END_VAR
VAR_OUTPUT
	ERROR_C : DWORD;
	ERROR_T : BYTE;
END_VAR
VAR
	FS : FILE_SERVER;
	FSD : FILE_SERVER_DATA;
	PT : NETWORK_BUFFER;
	UCB : UNI_CIRCULAR_BUFFER;
	ra : BOOL;
	trig_m_last : BOOL;
	dti_last : DT := DT#2070-02-06-06:28:15;
	enable_last : BOOL;
	fn_last : STRING;
	str : STRING(STRING_LENGTH);
	fn : STRING;
	init : BOOL;
	step: INT;
	idx : INT;
	log_state : USINT;
	color : BOOL;
	head: BOOL;
	n : INT;
END_VAR

(*
version 1.0		25. july. 2011
programmer		ks
tested by			ks

DLOG_STORE_FILE_HTML schreibt die DLOG Parameter in einen lokale Datei im HMTL-Format 

*)

X.DTI := DTI; (* Datum / Zeit eintragen *)
IF DTI <> dti_last THEN
	X.CLOCK_TRIG := TRUE;
	dti_last := DTI;
	X.STORE_TYPE := 4;
ELSE
	X.CLOCK_TRIG := FALSE;
END_IF;

IF X.ADD_HEADER = FALSE THEN (* wenn add-header und add-data gleichzeitig ansteht, dann add-data einen zyklus länger anstehen lassen *)
	X.ADD_DATA := FALSE;
END_IF;
X.ADD_HEADER := FALSE;

IF ENABLE THEN
	IF X.CLOCK_TRIG THEN
		fn := DT_TO_STRF(DTI, 0, FILENAME, 0); (* automatische Dateinamen generierung *)
		IF TRIG_T > 0 THEN (* automatischer Trigger *)
			ra := DT_TO_UDINT(DTI) MOD TRIG_T = 0;
		END_IF;
	ELSE
		ra := FALSE;
	END_IF;
	IF (TRIG_M AND NOT trig_m_last) OR ra OR X.ADD_DATA_REQ THEN (* manueller, automatischer oder externer Trigger *)
		X.ADD_DATA := TRUE; (* Daten loggen *)
	END_IF;
	IF NOT init THEN
		init := TRUE;
		X.ADD_HEADER := TRUE; (* Spaltenüberschriften übernehmen *)
	END_IF;
END_IF;
X.ADD_DATA_REQ := FALSE; (* externe Anforderung rücksetzen *)

IF (NOT ENABLE AND enable_last) OR (fn <> fn_last AND step > 0) THEN (* Neg. Flanke ENABLE - Log Stop *)
	fn_last := fn;
	X.UCB.D_HEAD := WORD#16#FF00;
	X.UCB.D_MODE := 1;
	UCB(DATA:=X.UCB); (* Element schreiben *)
	X.ADD_HEADER := TRUE; (* Spaltenüberschriften übernehmen *)
END_IF;

CASE step OF

00:	IF ENABLE THEN
		color := FALSE;
		head := FALSE;
		fn_last := fn;
		FSD.FILENAME := fn; (* Dateiname *)
		FSD.OFFSET := 0; (* Start bei Dateianfang *)
		FSD.AUTO_CLOSE := T#0s; (* Auto-Close *)
		step := 10;
	END_IF;

10:	(* Headerdaten schreiben *)
	str := CONCAT('<html><body><table ',HTML_TABLE);
         str := CONCAT(str,'><caption>');
         str := CONCAT(str,HTML_CAPTION);
         str := CONCAT(str,'</caption>');

	_STRING_TO_BUFFER(STR:=str, POS:=idx, PT:=ADR(PT.BUFFER), SIZE:=SIZEOF(PT.BUFFER));
	idx := idx + LEN(str);
	step := 20;

20:	IF log_state = 254 THEN
		log_state := 255;
		str := '</table></body></html>';
		_STRING_TO_BUFFER(STR:=str, POS:=idx, PT:=ADR(PT.BUFFER), SIZE:=SIZEOF(PT.BUFFER));
		idx := idx + LEN(str);
		step := 40; (* Daten schreiben *)

	ELSIF X.UCB.BUF_COUNT > 0 THEN (* Einträge vorhanden *)
		X.UCB.D_MODE := 10;
		UCB(DATA:=X.UCB); (* Element lesen , aber noch nicht entfernen *)

		IF X.UCB.D_HEAD = WORD#16#FF00 THEN (* LOG_STOP Command *)
			X.UCB.D_MODE := 11;
			UCB(DATA:=X.UCB); (* Element entfernen *)
			log_state := 254;

		ELSIF idx + LEN(X.UCB.D_STRING) + 120 < SIZEOF(PT) THEN (* Platz für Element vorhanden ? *)
			X.UCB.D_MODE := 11;
			UCB(DATA:=X.UCB); (* Element entfernen *)

			IF log_state = 0 THEN
				str := '<TR ';
				IF NOT head THEN
					str := CONCAT(str,HTML_TR_HEAD);
					head := TRUE;
				ELSIF color THEN
					str := CONCAT(str,HTML_TR_EVEN);
				ELSE
					str := CONCAT(str,HTML_TR_ODD);
				END_IF;
				str := CONCAT(str,'><TD>');
			ELSE
				str := '<TD>';
			END_IF;

			_STRING_TO_BUFFER(STR:=str, POS:=idx, PT:=ADR(PT.BUFFER), SIZE:=SIZEOF(PT.BUFFER));
			idx := idx + LEN(str);
			log_state := log_state + 1;

			_STRING_TO_BUFFER(STR:=X.UCB.D_STRING, POS:=idx, PT:=ADR(PT.BUFFER), SIZE:=SIZEOF(PT.BUFFER));
			idx := idx + LEN(X.UCB.D_STRING);
			n := n + 1;
			IF n = X.ID_MAX THEN
				n := 0;
				str := '</TD></TR>';
				color := NOT color;
				log_state := 0;
			ELSE
				str := '</TD>';
			END_IF;
			_STRING_TO_BUFFER(STR:=str, POS:=idx, PT:=ADR(PT.BUFFER), SIZE:=SIZEOF(PT.BUFFER));
			idx := idx + LEN(str);
		END_IF;
		step := 40; (* Daten schreiben *)
	END_IF;

40:	IF idx > 0 THEN (* Daten schreiben *)
		FSD.MODE := 3; (* create + write *)
		PT.SIZE := idx; (* Datenlänge eintragen *)
		idx := 0;
	END_IF;
	step := 60;

60:	IF FSD.MODE = 0 THEN
		IF log_state = 255 THEN
			log_state := 0;
			FSD.MODE := 5; (* Datei schliessen *)
			X.NEW_FILE := FSD.FILENAME;
			X.NEW_FILE_RTRIG := FALSE;
			step := 80;
		ELSE
			step := 20;
		END_IF;
	END_IF;

80:	IF FSD.MODE = 0 THEN (* Datei schliessen beendet *)
		X.NEW_FILE_RTRIG := TRUE;
		step := 0;
	END_IF;

END_CASE;

trig_m_last := TRIG_M;
enable_last := ENABLE;
FS(FSD:=FSD,PT:=PT); (* FILE_SERVER *)

ERROR_C := FSD.ERROR;
ERROR_T := SEL(FSD.ERROR > 0,0,1);

(* revision history
ks	25. july. 2011	rev 1.0
	original version

*)

END_FUNCTION_BLOCK

// oscat_network/POUs/DATA_LOG/DLOG_STORE_FILE_XML_1
FUNCTION_BLOCK DLOG_STORE_FILE_XML_1
VAR_IN_OUT
	X : DLOG_DATA;
END_VAR
VAR_INPUT
	ENABLE : BOOL;
	TRIG_M : BOOL;
	TRIG_T : UDINT;
	FILENAME : STRING;
	DTI : DT;
END_VAR
VAR_OUTPUT
	ERROR_C : DWORD;
	ERROR_T : BYTE;
END_VAR
VAR
	FS : FILE_SERVER;
	FSD : FILE_SERVER_DATA;
	PT : NETWORK_BUFFER;
	UCB : UNI_CIRCULAR_BUFFER;
	ra : BOOL;
	trig_m_last : BOOL;
	dti_last : DT := DT#2070-02-06-06:28:15;
	enable_last : BOOL;
	fn_last : STRING;
	str : STRING(STRING_LENGTH);
	fn : STRING;
	init : BOOL;
	step: INT;
	idx : INT;
	log_state : USINT;
	n : INT;
END_VAR

(*
version 1.0		25. july. 2011
programmer		ks
tested by			ks

DLOG_STORE_FILE_XML schreibt die DLOG Parameter in einen lokale Datei im XML-Format 

*)

X.DTI := DTI; (* Datum / Zeit eintragen *)
IF DTI <> dti_last THEN
	X.CLOCK_TRIG := TRUE;
	dti_last := DTI;
	X.STORE_TYPE := 3;
ELSE
	X.CLOCK_TRIG := FALSE;
END_IF;

IF X.ADD_HEADER = FALSE THEN (* wenn add-header und add-data gleichzeitig ansteht, dann add-data einen zyklus länger anstehen lassen *)
	X.ADD_DATA := FALSE;
END_IF;
X.ADD_HEADER := FALSE;

IF ENABLE THEN
	IF X.CLOCK_TRIG THEN
		fn := DT_TO_STRF(DTI, 0, FILENAME, 0); (* automatische Dateinamen generierung *)
		IF TRIG_T > 0 THEN (* automatischer Trigger *)
			ra := DT_TO_UDINT(DTI) MOD TRIG_T = 0;
		END_IF;
	ELSE
		ra := FALSE;
	END_IF;
	IF (TRIG_M AND NOT trig_m_last) OR ra OR X.ADD_DATA_REQ THEN (* manueller, automatischer oder externer Trigger *)
		X.ADD_DATA := TRUE; (* Daten loggen *)
	END_IF;
	IF NOT init THEN
		init := TRUE;
		X.ADD_HEADER := TRUE; (* Spaltenüberschriften übernehmen *)
	END_IF;
END_IF;
X.ADD_DATA_REQ := FALSE; (* externe Anforderung rücksetzen *)

IF (NOT ENABLE AND enable_last) OR (fn <> fn_last AND step > 0) THEN (* Neg. Flanke ENABLE - Log Stop *)
	fn_last := fn;
	X.UCB.D_HEAD := WORD#16#FF00;
	X.UCB.D_MODE := 1;
	UCB(DATA:=X.UCB); (* Element schreiben *)
	X.ADD_HEADER := TRUE; (* Spaltenüberschriften übernehmen *)
END_IF;

CASE step OF

00:	IF ENABLE THEN
		fn_last := fn;
		FSD.FILENAME := fn; (* Dateiname *)
		FSD.OFFSET := 0; (* Start bei Dateianfang *)
		FSD.AUTO_CLOSE := T#0s; (* Auto-Close *)
		step := 10;
	END_IF;

10:	(* Headerdaten schreiben *)
	str := '<?xml version="1.0" encoding="UTF-8"?><table>';
	_STRING_TO_BUFFER(STR:=str, POS:=idx, PT:=ADR(PT.BUFFER), SIZE:=SIZEOF(PT.BUFFER));
	idx := idx + LEN(str);
	step := 20;

20:	IF log_state = 254 THEN
		log_state := 255;
		str := '</table>';
		_STRING_TO_BUFFER(STR:=str, POS:=idx, PT:=ADR(PT.BUFFER), SIZE:=SIZEOF(PT.BUFFER));
		idx := idx + LEN(str);
		step := 40; (* Daten schreiben *)

	ELSIF X.UCB.BUF_COUNT > 0 THEN (* Einträge vorhanden *)
		X.UCB.D_MODE := 10;
		UCB(DATA:=X.UCB); (* Element lesen , aber noch nicht entfernen *)

		IF X.UCB.D_HEAD = WORD#16#FF00 THEN (* LOG_STOP Command *)
			X.UCB.D_MODE := 11;
			UCB(DATA:=X.UCB); (* Element entfernen *)
			log_state := 254;

		ELSIF idx + LEN(X.UCB.D_STRING) + 120 < SIZEOF(PT) THEN (* Platz für Element vorhanden ? *)
			X.UCB.D_MODE := 11;
			UCB(DATA:=X.UCB); (* Element entfernen *)

			IF log_state = 0 THEN
				str := '<row><entry>';
			ELSE
				str := '<entry>';
			END_IF;

			_STRING_TO_BUFFER(STR:=str, POS:=idx, PT:=ADR(PT.BUFFER), SIZE:=SIZEOF(PT.BUFFER));
			idx := idx + LEN(str);
			log_state := log_state + 1;

			_STRING_TO_BUFFER(STR:=X.UCB.D_STRING, POS:=idx, PT:=ADR(PT.BUFFER), SIZE:=SIZEOF(PT.BUFFER));
			idx := idx + LEN(X.UCB.D_STRING);

			n := n + 1;
			IF n = X.ID_MAX THEN
				n := 0;
				str := '</entry></row>';
				log_state := 0;
			ELSE
				str := '</entry>';
			END_IF;
			_STRING_TO_BUFFER(STR:=str, POS:=idx, PT:=ADR(PT.BUFFER), SIZE:=SIZEOF(PT.BUFFER));
			idx := idx + LEN(str);
		END_IF;
		step := 40; (* Daten schreiben *)
	END_IF;

40:	IF idx > 0 THEN (* Daten schreiben *)
		FSD.MODE := 3; (* create + write *)
		PT.SIZE := idx; (* Datenlänge eintragen *)
		idx := 0;
	END_IF;
	step := 60;

60:	IF FSD.MODE = 0 THEN
		IF log_state = 255 THEN
			log_state := 0;
			FSD.MODE := 5; (* Datei schliessen *)
			X.NEW_FILE := FSD.FILENAME;
			X.NEW_FILE_RTRIG := FALSE;
			step := 80;
		ELSE
			step := 20;
		END_IF;
	END_IF;

80:	IF FSD.MODE = 0 THEN (* Datei schliessen beendet *)
		X.NEW_FILE_RTRIG := TRUE;
		step := 0;
	END_IF;

END_CASE;

trig_m_last := TRIG_M;
enable_last := ENABLE;
FS(FSD:=FSD,PT:=PT); (* FILE_SERVER *)

ERROR_C := FSD.ERROR;
ERROR_T := SEL(FSD.ERROR > 0,0,1);

(* revision history
ks	25. july. 2011	rev 1.0
	original version

*)

END_FUNCTION_BLOCK

// oscat_network/POUs/DATA_LOG/DLOG_STORE_RRD_1
FUNCTION_BLOCK DLOG_STORE_RRD_1
VAR_IN_OUT
	X : DLOG_DATA;
END_VAR
VAR_INPUT
	ENABLE : BOOL;
	TRIG_M : BOOL;
	TRIG_T : UDINT;
	URL : STRING(STRING_LENGTH);
	DTI : DT;
	SEP : BYTE;
	DNS_IP4 : DWORD;
	TIMEOUT : TIME;
END_VAR
VAR_OUTPUT
	ERROR_C : DWORD;
	ERROR_T : BYTE;
END_VAR
VAR
	UCB : UNI_CIRCULAR_BUFFER;
	IP_C : IP_C; (* IP_Control Verwaltungsstruktur *)
	S_BUF : NETWORK_BUFFER;
	R_BUF : NETWORK_BUFFER;
	URL_DATA : url;
	DNS_CLIENT : DNS_CLIENT;
	HTTP_GET : HTTP_GET;
	IPC : IP_CONTROL;

	ra : BOOL;
	trig_m_last : BOOL;
	dti_last : DT := DT#2070-02-06-06:28:15;
	step: INT;
	sep_char : STRING(1);
	n : INT;
END_VAR

(*
version 1.2		26. july. 2011
programmer		ks
tested by			ks

DLOG_STORE_RRD der Baustein übergibt die DLOG Parameter an einen RoundRobinDatabase-Server
*)

X.DTI := DTI; (* Datum / Zeit eintragen *)
IF DTI <> dti_last THEN
	X.CLOCK_TRIG := TRUE;
	dti_last := DTI;
	X.STORE_TYPE := 1;
ELSE
	X.CLOCK_TRIG := FALSE;
END_IF;

X.ADD_DATA := FALSE;

IF ENABLE THEN
	IF X.CLOCK_TRIG THEN
		IF TRIG_T > 0 THEN (* automatischer Trigger *)
			ra := DT_TO_UDINT(DTI) MOD TRIG_T = 0;
		END_IF;
	ELSE
		ra := FALSE;
	END_IF;
	IF (TRIG_M AND NOT trig_m_last) OR ra OR X.ADD_DATA_REQ THEN (* manueller, automatischer oder externer Trigger *)
		X.ADD_DATA := TRUE; (* Daten loggen *)
	END_IF;
END_IF;
X.ADD_DATA_REQ := FALSE; (* externe Anforderung rücksetzen *)

CASE step OF

00:	IF ENABLE THEN
		URL_DATA:=STRING_TO_URL(STR:=URL,DEFAULT_PROTOCOL:='',DEFAULT_PATH:=''); (* URL zerlegen *)
		sep_char := CHR_TO_STRING(SEP);
		ERROR_T := 0;
		ERROR_C := 0;
		step := 20;
	END_IF;

20:	IF X.UCB.BUF_COUNT >= X.ID_MAX THEN (* Einträge vorhanden *)
		n := 1;
		WHILE n <= X.ID_MAX DO
			X.UCB.D_MODE := 12; (* Element lesen und löschen *)
			UCB(DATA:=X.UCB);
			IF n < X.ID_MAX THEN (* Trennzeichen hinzufügen *)
				X.UCB.D_STRING := CONCAT(X.UCB.D_STRING,sep_char);
			END_IF;
			IF LEN(X.UCB.D_STRING) + LEN(URL_DATA.QUERY) <= STRING_LENGTH THEN
				URL_DATA.QUERY := CONCAT(URL_DATA.QUERY,X.UCB.D_STRING); (* Query mit LOG-Daten ergänzen *)
				step :=40;
			ELSE
				ERROR_T := 4; (* LOG-Daten können nicht in URL gepackt werden *)
				ERROR_C := 1;
				step := 0;
			END_IF;
			n := n + 1;
		END_WHILE;;
	END_IF;

40:	IF DNS_CLIENT.DONE THEN
		step := 60;
	ELSIF (DNS_CLIENT.ERROR > 0) THEN
		ERROR_C := DNS_CLIENT.ERROR; (* Fehlerbehandlung *)
		ERROR_T := 1;
		step := 100;
	END_IF;

60:	IF HTTP_GET.DONE THEN
		n := HTTP_GET.BODY_START;
		IF R_BUF.BUFFER[n] <> 48 THEN (* ASCII '0' *)
			ERROR_C := 1;
			ERROR_T := 3;
		END_IF;
		step := 100;

	ELSIF HTTP_GET.ERROR > 0 THEN (* Fehlerbehandlung *)
		ERROR_C := HTTP_GET.ERROR;
		ERROR_T := 2;
		step := 100;
	END_IF;

100:	IF (NOT HTTP_GET.DONE) THEN (* UNLOCK HTTP DATA *)
		step := SEL(ERROR_T = 0, 120,0);
	END_IF;

120:	IF NOT ENABLE THEN
		X.UCB.D_MODE := 99;
		UCB(DATA:=X.UCB); (* Buffer löschen *)
		step := 0;
	END_IF;

END_CASE;

HTTP_GET(IP_C:=IP_C,S_BUF:=S_BUF,R_BUF:=R_BUF,IP4:=DNS_CLIENT.IP4,GET:=step=60,MODE:=2,UNLOCK_BUF:=step=100,URL_DATA:=URL_DATA); (* HTTP_GET *)
DNS_CLIENT(IP_C:=IP_C, S_BUF:=S_BUF, R_BUF:=R_BUF, DOMAIN:=URL_DATA.DOMAIN, IP4_DNS:= DNS_IP4, ACTIVATE:=step=40); (* DNS-Client *)
IPC(IP:= 0, PORT:= 0 , TIME_OUT:= TIMEOUT, IP_C:= IP_C, S_BUF:= S_BUF, R_BUF:= R_BUF); (* IP_CONTROL *)

trig_m_last := TRIG_M;

(* revision history
ks	01. jan. 2011	rev 1.0
	original version

ks	13. may. 2011	rev 1.1
	ADD_DATA_REQ hinzugefügt

ks	26. july. 2011	rev 1.2
	code optimierung D_MODE 12 und bessere fehlerauswertung
*)

END_FUNCTION_BLOCK

// oscat_network/POUs/NETWORK/HTTP_GET
FUNCTION_BLOCK HTTP_GET
VAR_IN_OUT
	URL_DATA : url;
	IP_C : IP_C; (* IP_Control Verwaltungsstruktur *)
	S_BUF : NETWORK_BUFFER;
	R_BUF : NETWORK_BUFFER;
END_VAR
VAR_INPUT
	IP4 : DWORD;
	GET : BOOL;
	MODE : BYTE := BYTE#2;
	UNLOCK_BUF : BOOL;
END_VAR
VAR_OUTPUT
	HTTP_STATUS : STRING;
	HEADER_START : UINT; (* HTTP Header (Message Header) *)
	HEADER_STOP : UINT; (* HTTP Header (Message Header) *)
	BODY_START : UINT; (* Message Body *)
	BODY_STOP : UINT; (* Message Body *)
	DONE : BOOL;
	ERROR : DWORD;
END_VAR
VAR
	READ_HTTP :	READ_HTTP;
	IP_FIFO : IP_FIFO;
	ip_state : BYTE;
	ip_id : BYTE;
	get_last : BOOL;
	ip4_stored : DWORD;
	state : INT;
	i : INT;
	http_1_1_host : BOOL;
	total_size : INT;
	text : STRING(STRING_LENGTH);
	delimiter2b : STRING(2);
	delimiter4b : STRING(4);
	del_end : STRING(4);
	del_pos : INT;
	idx : INT;
	rcv_timeout : BOOL;
	con_rdce : BOOL;

	(*LOG_MSG : LOG_MSG;
	_debug_enable : BOOL := TRUE;*)

END_VAR

(*

version 1.3	12. apr. 2011
programmer 	ks
tested by		ks

HTTP_GET führt eine HTTP Abfrage einer Web-Seite bei einem WEB_Server durch, und stellt die Daten ausbereitet zu verfügung
*)

CASE state OF
00:	IF GET AND NOT GET_LAST THEN (* auf positive Flanke SET warten *)
		state := 10;
		ip4_stored := IP4; (* aktuelle IP4 speichern *)
		DONE := FALSE;
		total_size := 0;
		HEADER_START := UINT#0;
		HEADER_STOP := UINT#0;
		BODY_START := UINT#0;
		BODY_STOP := UINT#0;
		HTTP_STATUS := '';
		ERROR := DWORD#0;
		ip_state := BYTE#1; (* Anmelden *)
		delimiter2b := '$0D$0A';
		delimiter4b := '$0D$0A$0D$0A';
	        	(*####################  DEBUG-MESSAGE  ###################################*)
		(*IF _debug_enable THEN
	       		LOG_CL.NEW_MSG := 'HTTP: S00 START /IP_ID ~4';
	            	LOG_CL.PRINTF[4]  := BYTE_TO_STRING(IP_ID);
	            	LOG_MSG();
	        	END_IF;*)
	        	(*########################################################################*)
	END_IF;

10:	IF ip_state = BYTE#3 THEN (* Bei IP_Control anmelden und auf freigabe warten *)
		idx := 0;
		text := CONCAT('GET ',URL_DATA.PATH);
		_STRING_TO_BUFFER(STR:=text,POS:=idx,PT:=ADR(S_BUF.BUFFER),SIZE:=SIZEOF(S_BUF.BUFFER)); (* GET path in buffer kopieren *)
		idx := idx + LEN(text);

		IF LEN(URL_DATA.QUERY) > 0 THEN
			S_BUF.BUFFER[idx] := 63; (* ASCII '?' *)
			idx := idx + 1;
			_STRING_TO_BUFFER(STR:=URL_DATA.QUERY,POS:=idx,PT:=ADR(S_BUF.BUFFER),SIZE:=SIZEOF(S_BUF.BUFFER)); (* QUERY in buffer kopieren *)
			idx := idx + LEN(URL_DATA.QUERY);
		END_IF;

		IF MODE >= BYTE#2 THEN (* gewünschte HTTP Version uebergeben *)
			text := ' HTTP/1.1';
		ELSE
			text := ' HTTP/1.0';
		END_IF;
		text := CONCAT(text,delimiter2b);
		_STRING_TO_BUFFER(STR:=text,POS:=idx,PT:=ADR(S_BUF.BUFFER),SIZE:=SIZEOF(S_BUF.BUFFER)); (* HTTP Version in buffer kopieren *)
		idx := idx + LEN(text);

		IF MODE = BYTE#1 THEN (* HTTP/1.0 mit persistenter Verbindung gewünscht *)
			text := CONCAT('Connection: Keep-Alive',delimiter2b); (* workaround für pcworx -> kein $0D$0A als Stringkonstante möglich *)
		ELSIF MODE = BYTE#3 THEN (* HTTP/1.1 ohne persistenter Verbindung gewünscht *)
			text := CONCAT('Connection: Close',delimiter2b); (* workaround für pcworx -> kein $0D$0A als Stringkonstante möglich *)
		ELSE
			text := '';
		END_IF;
		text := CONCAT(text,URL_DATA.HEADER);
		_STRING_TO_BUFFER(STR:=text,POS:=idx,PT:=ADR(S_BUF.BUFFER),SIZE:=SIZEOF(S_BUF.BUFFER)); (* HTTP Version in buffer kopieren *)
		idx := idx + LEN(text);

		text := CONCAT('Host: ',URL_DATA.DOMAIN);
		text := CONCAT(text,delimiter4b); (* workaround für pcworx -> kein $0D$0A als Stringkonstante möglich *)
		_STRING_TO_BUFFER(STR:=text,POS:=idx,PT:=ADR(S_BUF.BUFFER),SIZE:=SIZEOF(S_BUF.BUFFER)); (* HTTP Host in buffer kopieren *)
		idx := idx + LEN(text);

		(* IP Datenverkehr einrichten *)
		IF URL_DATA.PORT = WORD#0 THEN
			IP_C.C_PORT := WORD#80; (* Standard-Portnummer verwenden *)
		ELSE
			IP_C.C_PORT := URL_DATA.PORT; (* Portnummer aus URL verwenden *)
		END_IF;

		IP_C.C_IP := ip4_stored; (* IP eintragen *)
		IP_C.C_MODE := BYTE#0; (* Mode: TCP+AKTIV+PORT+IP *)
		IP_C.C_ENABLE := TRUE; (* Verbindungsaufbau freigeben *)
		IP_C.TIME_RESET := TRUE; (* Zeitueberwachung rücksetzen *)
		IP_C.R_OBSERVE := TRUE; (* Datenempfang ueberwachen *)
		S_BUF.SIZE := INT_TO_UINT(idx); (* Sendelänge eintragen *)
		R_BUF.SIZE := UINT#0; (* Empfangslänge rücksetzen *)

		state := 30;
	        	(*####################  DEBUG-MESSAGE  ###################################*)
	        	(*IF _debug_enable THEN
	        		LOG_CL.NEW_MSG := 'HTTP: S20 SEND /IP_ID ~4';
	            	LOG_CL.PRINTF[4]  := BYTE_TO_STRING(IP_ID);
	            	LOG_MSG();
	        	END_IF;*)
	        	(*########################################################################*)
	END_IF;

30:	rcv_timeout := (IP_C.ERROR AND DWORD#16#0000_FF00) = DWORD#16#0000_FF00;
	con_rdce :=     (IP_C.ERROR AND DWORD#16#FD00_0000) = DWORD#16#FD00_0000;

	IF S_BUF.SIZE = UINT#0 THEN
		IF total_size = 0 THEN
			IF R_BUF.SIZE > UINT#15 THEN; (* länge der empfangenen Daten prüfen *)

				(* HTTP HEADER Ende suchen -> durch $0D$A$0D$A erkennbar bei DEC RT-11,CP/M,MS-DOS,Windows *)
				del_end := '$0D$0A$0D$0A';
				del_pos := BUFFER_SEARCH(PT:=ADR(R_BUF.BUFFER),SIZE:=R_BUF.SIZE,STR:=del_end,POS:=0,IGN:=FALSE);

				(* kein Ende gefunden ? -> andere Ende-Codierung suchen *)
				IF del_pos = 0 THEN
					del_end := '$0A$0A';
					(* HTTP HEADER Ende suchen -> durch $0A$0A erkennbar bei Multics, Unix-Derivate,Mac OS X *)
					del_pos := BUFFER_SEARCH(PT:=ADR(R_BUF.BUFFER),SIZE:=R_BUF.SIZE,STR:=del_end,POS:=0,IGN:=FALSE);
				END_IF;

				IF del_pos > 0 THEN
					HEADER_START := UINT#0;
					HEADER_STOP := INT_TO_UINT(del_pos + LEN(del_end) - 1);
					TOTAL_SIZE := -1; (* HTTP Header empfangen aber noch keine gesamtlänge bekannt *)
				END_IF;
		                	(*####################  DEBUG-MESSAGE  ###################################*)
		                	(*IF _debug_enable THEN
		                   	LOG_CL.NEW_MSG := 'HTTP: S20 HEADER_START ~1 / HEADER_STOP ~2/IP_ID ~4';
		                   	LOG_CL.PRINTF[4]  := BYTE_TO_STRING(IP_ID);
		                   	LOG_CL.PRINTF[1]  := UINT_TO_STRING(HEADER_START);
		                   	LOG_CL.PRINTF[2]  := UINT_TO_STRING(HEADER_STOP);
		                   	LOG_MSG();
		                	END_IF;*)
		                	(*########################################################################*)

				(* HTTP Statuscode auswerten: (kann 1.0 oder 1.1 sein *)
				READ_HTTP(size:=HEADER_STOP,pos:=0,SRC:='',pt:=R_BUF.BUFFER);

				i := LEN(READ_HTTP.READ_HTTP);
				IF i > 7 THEN
					(* HTTP Version von HOST auswerten 1.0 oder 1.1 *)
					text:=MID(READ_HTTP.READ_HTTP,1,3);
					http_1_1_host := text = '1';

					(* Code und Meldung isolieren *)
					HTTP_STATUS := RIGHT(READ_HTTP.READ_HTTP,i-4);
				END_IF;

				(* positive HTTP Anfrage ? *)
				IF FIND(HTTP_STATUS,'200') > 0 THEN

					(* 'Content-Length: Wert einlesen auswerten *)
					READ_HTTP(size:=HEADER_STOP,pos:=0,SRC:='CONTENT-LENGTH',pt:=R_BUF.BUFFER);
					text:=READ_HTTP.READ_HTTP;

					IF LEN(text) >= 1 THEN
						IF IS_NUM(str:=text) THEN
							(* erwartete gesamtmenge an Bytes berechnen *)
							total_size := STRING_TO_INT(text) + UINT_TO_INT(HEADER_STOP) + 1;
                           					(*####################  DEBUG-MESSAGE  ###################################*)
                           					(*IF _debug_enable THEN
                              					LOG_CL.NEW_MSG := 'HTTP: S20 HEADER ~1, BODY ~2 TOTAL ~3 /IP_ID ~4';
                             					LOG_CL.PRINTF[4]  := BYTE_TO_STRING(IP_ID);
                               					LOG_CL.PRINTF[1]  := UINT_TO_STRING(HEADER_STOP);
                               					LOG_CL.PRINTF[2]  := INT_TO_STRING(TOTAL_SIZE-UINT_TO_INT(HEADER_STOP));
                               					LOG_CL.PRINTF[3]  := INT_TO_STRING(TOTAL_SIZE);
                              					LOG_MSG();
                          					END_IF;*)
                          					(*########################################################################*)
						END_IF;
					END_IF;
				ELSE
					ERROR := DWORD#16#000000FC; (* Fehler durch HTTP-Statuscodes *)
				END_IF;
			END_IF;
		(* 1. bei bekannter Content-Length wird nach erhalt der erwartenen Daten die verbindung beendet *)
		(* 2. bei persistenter Verbindung muss bei unbekannter Datenmenge auf Receive-Timeout gewartet werden *)
		(* 3. wenn nach datenempfang die verbindung vom host unterbrochen wird *)
		ELSIF (R_BUF.SIZE >= INT_TO_UINT(total_size)) OR
			(R_BUF.SIZE > UINT#0 AND total_size < 0 AND ((rcv_timeout OR con_rdce) OR (IP_C.C_STATE = BYTE#1))) THEN

			IF R_BUF.SIZE - 1 > HEADER_STOP THEN (* BODY Daten vorhanden *)
				BODY_START := HEADER_STOP + UINT#1;
				BODY_STOP := R_BUF.SIZE - 1;
		                	(*####################  DEBUG-MESSAGE  ###################################*)
		                	(*IF _debug_enable THEN
		                   	LOG_CL.NEW_MSG := 'HTTP: S20 BODY ~1, START ~2 END ~3 /IP_ID ~4';
		                   	LOG_CL.PRINTF[4]  := BYTE_TO_STRING(IP_ID);
		                   	LOG_CL.PRINTF[1]  := UINT_TO_STRING(HEADER_STOP);
		                   	LOG_CL.PRINTF[2]  := UINT_TO_STRING(BODY_START);
		                   	LOG_CL.PRINTF[3]  := UINT_TO_STRING(BODY_STOP);
		                   	LOG_MSG();
		               	END_IF;*)
		               	(*########################################################################*)
			END_IF;

			DONE := TRUE;
			IP_C.C_ENABLE := FALSE; (* Verbindung abbauen *)
			state := 40;
            		(*####################  DEBUG-MESSAGE  ###################################*)
            		(*IF _debug_enable THEN
                			LOG_CL.NEW_MSG := 'HTTP: S30 OK /IP_ID ~4';
                			LOG_CL.PRINTF[4]  := BYTE_TO_STRING(IP_ID);
                			LOG_MSG();
            		END_IF;*)
            		(*########################################################################*)
		END_IF;
	END_IF;

	IF IP_C.ERROR <> DWORD#0 THEN
		(* bei unbekannter Content-size ist nicht bekannt ob bzw wieviele Telegramme noch folgen werden *)
		(* darum wird nach receive-timeout oder Remote disconnect error der fehler wieder ausgefiltert (logischer fehler) *)
		IF rcv_timeout AND DONE THEN
			IP_C.ERROR := IP_C.ERROR AND DWORD#16#FFFF_00FF; (* Fehler wieder rücksetzen *)
		ELSIF con_rdce AND DONE THEN
			IP_C.ERROR := IP_C.ERROR AND DWORD#16#00FF_FFFF; (* Fehler wieder rücksetzen *)
		ELSE
			ERROR := IP_C.ERROR;
		END_IF;
	END_IF;

	IF ERROR > DWORD#0 THEN
		IP_C.C_ENABLE := FALSE; (* Verbindungsaufbau sperren *)
		state := 40;
	        	(*####################  DEBUG-MESSAGE  ###################################*)
	        	(*IF _debug_enable THEN
	            	LOG_CL.NEW_MSG := 'HTTP: S30 ERROR ~1 /IP_ID ~4';
	            	LOG_CL.PRINTF[1]  := DWORD_TO_STRING(ERROR);
	            	LOG_CL.PRINTF[4]  := BYTE_TO_STRING(IP_ID);
	            	LOG_MSG();
	        	END_IF;*)
	        	(*########################################################################*)
	END_IF;

40:	IF (UNLOCK_BUF OR NOT DONE) THEN (* Warten auf Release und Verbindung beendet -> IP_ID vom Stack nehmen *)
		IP_STATE := BYTE#4; (* Abmelden *)
		DONE := FALSE;
		state := 0;
	END_IF;
END_CASE;

get_last := GET; (* letzten Status sichern zur Flankenerkennung *)

IP_FIFO(FIFO:=IP_C.FIFO,STATE:=ip_state,ID:=ip_id); (* IP_FIFO *)

(* revision history
ks	18. oct. 2008	rev 1.0
	original version

ks	20. oct. 2009	rev 1.1
	Fehler bei body-suche bei $0a$0a korrigiert,Codeoptimierung,
	new VAR del_pos , del_end (Networkbuffer und Buffer-funktionen auf Basis 0)

ks	28. oct. 2009	rev 1.2
	über url.header können zusätzliche header-infos übergeben werden

ks	12. apr. 2011	rev 1.3
	verbesserte fehlererkennung und fehlerkorrektur bei buffer_to_string
*)

END_FUNCTION_BLOCK

// oscat_network/POUs/NETWORK/READ_HTTP
FUNCTION_BLOCK READ_HTTP
VAR_INPUT
	SIZE : UINT;
	POS : INT;
	SRC : STRING;
END_VAR
VAR_IN_OUT
	PT : NW_BUF_LONG;
END_VAR
VAR_OUTPUT
	READ_HTTP : STRING(STRING_LENGTH);
END_VAR
VAR
	index : INT;
	s1 : INT;
	e1 : INT;
	stop : INT;
END_VAR

(*

version 1.1 20. oct. 2009
programmer 	ks
tested by	ks

READ_HTTP wertet die Informationen einer HTTP-Request aus, und stellt die Daten zu Verfügung.
*)

stop := UINT_TO_INT(SIZE) - 1;

IF LEN(SRC) = 0 THEN
	(* wenn kein Suchbegriff vorhanden ist, dann den HTTP-STATUS auswerten *)
	SRC := 'HTTP/'; (* neuer Suchbegriff *)
ELSE
	(* gesuchten Parametertext ergänzen *)
	SRC := CONCAT(SRC,': ');
END_IF;

s1 := BUFFER_SEARCH(pt:=ADR(PT),SIZE:=SIZE,STR:=SRC,POS:=POS,IGN:=TRUE);

IF s1 >= 0 THEN (* Text found *)
	e1 := s1;

	(* search start of line *)
	index := s1 - 1;
	WHILE (index > 0) DO
		IF pt[index] < BYTE#32 THEN EXIT; END_IF;
		s1 := s1 - 1;
		index := index - 1;
	END_WHILE;

	(* search end of line *)
	index := e1 + 1;
	WHILE (index <= stop) DO
		IF pt[index] < BYTE#32 THEN EXIT; END_IF;
		e1 := e1 + 1;
		index := index + 1;
	END_WHILE;

	s1 := s1 + LEN(SRC); (* 'suchbegriff: ' nicht mitkopieren *)

	(* copy string *)
	READ_HTTP := BUFFER_TO_STRING(PT:=ADR(PT),SIZE:=SIZE,START:=s1,STOP:=e1);
ELSE
	READ_HTTP := '';
END_IF;

(* revision history

ks	18. oct. 2008	rev 1.0
	original version

ks	20. oct. 2009	rev 1.1
	Networkbuffer und Buffer-funktionen auf Basis 0

*)

END_FUNCTION_BLOCK

// oscat_network/POUs/DATA_LOG/DLOG_STRING_1
FUNCTION_BLOCK DLOG_STRING_1
VAR_IN_OUT
	X : DLOG_DATA;
END_VAR
VAR_INPUT
	STR : STRING;
	COLUMN : STRING(40);
END_VAR
VAR_OUTPUT
END_VAR
VAR
	UCB : UNI_CIRCULAR_BUFFER;
	init : BOOL;
	id : WORD;
	str_last : STRING;
END_VAR

(*
version 1.2		25. july. 2011
programmer		ks
tested by			ks

DLOG_STRING legt den STRING im FIFO-RING-Buffer ab um diesen mit den Baustein DLOG_STORE_*  aufzuzeichnen
*)

IF NOT init THEN
	init := TRUE;
	X.ID_MAX := X.ID_MAX + 1;
	id := WORD#16#0101; (* Quelltype STRING , Zieltype STRING *)
END_IF;

IF X.ADD_HEADER THEN
	X.UCB.D_STRING := COLUMN;
	X.UCB.D_HEAD := id;
	X.UCB.D_MODE := 1;
	UCB(DATA:=X.UCB); (* Daten eintragen *)
ELSIF X.ADD_DATA THEN
	X.UCB.D_STRING := str_last;
	X.UCB.D_HEAD := id;
	X.UCB.D_MODE := 1;
	UCB(DATA:=X.UCB); (* Daten eintragen *)
END_IF;
str_last := STR;

(* revision history
ks	01. jan. 2011	rev 1.0
	original version

ks	17. may. 2011	rev 1.1
	COLUMN STRING(40)

ks	25. july.   2011	rev 1.2
	neue head information
*)

END_FUNCTION_BLOCK

// oscat_network/POUs/DATA_LOG/UNI_CIRCULAR_BUFFER_1
FUNCTION_BLOCK UNI_CIRCULAR_BUFFER_1
VAR_IN_OUT
	DATA : UNI_CIRCULAR_BUFFER_DATA;
END_VAR
VAR_TEMP
	tmp_dw : DWORD;
	pTmp : POINTER TO BYTE;
	n : INT;
	n1 : INT;
	n2 : INT;
	x: BYTE;
	buf_totalsize : UINT;
END_VAR
VAR CONSTANT
	HeaderSize : INT := 4;
END_VAR
VAR
	cnt : UINT;
	mode_last : INT;

	(*LOG_MSG : LOG_MSG;
	_debug_enable : BOOL := FALSE;*)
END_VAR

(*
version 1.1		25. july. 2011
programmer		ks
tested by			ks

UNI_CIRCULAR_BUFFER ist ein FIFO-RING-Buffer der verschiedene Datenelemente als Byte-Array aufnehmen kann.
*)

CASE DATA.D_MODE OF

01:	x := WORD_TO_BYTE(DATA.D_HEAD); (* nur rechtes byte auswerten *)
	CASE x OF
	01:	cnt := LEN(DATA.D_STRING); (* String verarbeiten *)
		pTmp := ADR(DATA.D_STRING);
	02:	cnt := 4; (* Real verarbeiten *)
		pTmp := ADR(DATA.D_REAL);
	03:	cnt := 4; (* DWORD verarbeiten *)
		pTmp := ADR(DATA.D_DWORD);
	ELSE
		cnt := 0;
	END_CASE;

	(* ------ Daten in buffer eintragen ------ *)
	buf_totalsize := SIZEOF(DATA.BUF);

	IF (cnt + HeaderSize) > (buf_totalsize - DATA.BUF_SIZE) THEN (* genug Speicher frei ? *)
		RETURN;
	END_IF;

	mode_last := DATA.D_MODE;
	tmp_dw := SHL(WORD_TO_DWORD(DATA.D_HEAD),16) OR UINT_TO_DWORD(cnt);

	(* Header in Buffer eintragen *)
	n1 := 0;
	REPEAT
		n2 := MIN(HeaderSize - n1, buf_totalsize - DATA._Last);
		FOR n := 1 TO n2 DO
			tmp_dw := ROL(tmp_dw,8);
			data.BUF[DATA._Last] := DWORD_TO_BYTE(tmp_dw);
			DATA._Last := DATA._Last + 1;
		END_FOR;
		IF DATA._Last >= buf_totalsize THEN
			DATA._Last := 0;
		END_IF
		n1 := n1 + n2;
	UNTIL n1 >= HeaderSize
	END_REPEAT;

	(* Daten in Buffer eintragen *)
	n1 := 0;
	REPEAT
		n2 := MIN(cnt - n1, buf_totalsize - DATA._Last);
		FOR n := 1 TO n2 DO
			data.BUF[DATA._Last] := pTmp^;
			pTmp := pTmp + 1;
			DATA._Last := DATA._Last + 1;
		END_FOR;
		IF DATA._Last >= buf_totalsize THEN
			DATA._Last := 0;
		END_IF
		n1 := n1 + n2;
	UNTIL n1 >= cnt
	END_REPEAT;

	DATA.BUF_SIZE := DATA.BUF_SIZE + cnt + HeaderSize;
	DATA.BUF_COUNT := DATA.BUF_COUNT + 1;
	DATA.BUF_USED := UINT_TO_USINT(100 * DATA.BUF_SIZE / buf_totalsize); (* benützer Speicher in % *)
	DATA.D_MODE := 0;

	(*####################  DEBUG-MESSAGE  ###################################*)
	(*IF _debug_enable THEN
		LOG_CL.NEW_MSG := 'RP: ADD /HEAD ~1 / SIZE ~2 / CNT ~3 / >~4<';
		LOG_CL.PRINTF[1] := DWORD_TO_STRH(DATA.D_HEAD);
		LOG_CL.PRINTF[2] := UINT_TO_STRING(cnt);
		LOG_CL.PRINTF[3] := UINT_TO_STRING(DATA.BUF_COUNT);
		CASE x OF
		01:	LOG_CL.PRINTF[4] := DATA.D_STRING;
		02:	LOG_CL.PRINTF[4] := REAL_TO_STRING(DATA.D_REAL);
		03:	LOG_CL.PRINTF[4] := DWORD_TO_STRH(DATA.D_DWORD);
		ELSE
			LOG_CL.PRINTF[4] := '';
		END_CASE;
		LOG_MSG();
	END_IF;*)
	(*########################################################################*)

10..12:	(* ------ Daten aus buffer auslesen und optional löschen ------ *)
		(* 10 = nur lesen / 11 = löschen nach lesen / 12 = lesen und löschen *)
	IF DATA.D_MODE <> 11 THEN
		IF DATA.BUF_COUNT = 0 THEN RETURN; END_IF;
		buf_totalsize := SIZEOF(DATA.BUF);
		DATA._GetEnd := DATA._First;(* index des ältesten eintrags merken *)
		mode_last := DATA.D_MODE;
	
		(* Header aus Buffer lesen *)
		n1 := 0;
		tmp_dw := 0;
		REPEAT
			n2 := MIN(HeaderSize - n1, buf_totalsize - DATA._GetEnd);
			FOR n := 1 TO n2 DO
				tmp_dw := ROL(tmp_dw,8) OR BYTE_TO_DWORD(data.BUF[DATA._GetEnd]);
				DATA._GetEnd := DATA._GetEnd + 1;
			END_FOR;
			IF DATA._GetEnd >= buf_totalsize THEN
				DATA._GetEnd := 0;
			END_IF
			n1 := n1 + n2;
		UNTIL n1 >= HeaderSize
		END_REPEAT;
	
		DATA._GetStart := DATA._GetEnd;
		cnt := DWORD_TO_UINT(tmp_dw AND 16#0000_FFFF);
		DATA.D_HEAD := DWORD_TO_WORD(SHR(tmp_dw,16));
	
		x := WORD_TO_BYTE(DATA.D_HEAD); (* nur rechtes byte auswerten *)
		CASE x OF
		01:	pTmp := ADR(DATA.D_STRING); (* String verarbeiten *)
		02:	pTmp := ADR(DATA.D_REAL); (* Real verarbeiten *)
		03:	pTmp := ADR(DATA.D_DWORD); (* DWORD verarbeiten *)
		END_CASE;
	
		(* Daten aus Buffer lesen *)
		n1 := 0;
		REPEAT
			n2 := MIN(cnt - n1, buf_totalsize - DATA._GetEnd);
			FOR n := 1 TO n2 DO
				pTmp^ := data.BUF[DATA._GetEnd];
				pTmp := pTmp + 1;
				DATA._GetEnd := DATA._GetEnd + 1;
			END_FOR;
			IF DATA._GetEnd >= buf_totalsize THEN
				DATA._GetEnd := 0;
			END_IF
			n1 := n1 + n2;
		UNTIL n1 >= cnt
		END_REPEAT;
		IF x = 1 THEN
			pTmp^ := 0; (* String terminieren *)
		END_IF;
		DATA.D_MODE := 0;
	
		(*####################  DEBUG-MESSAGE  ###################################*)
		(*IF _debug_enable THEN
			LOG_CL.NEW_MSG := 'RP: READ /HEAD ~1 / SIZE ~2 / CNT ~3 / >~4<';
			LOG_CL.PRINTF[1] := DWORD_TO_STRH(DATA.D_HEAD);
			LOG_CL.PRINTF[2] := UINT_TO_STRING(cnt);
			LOG_CL.PRINTF[3] := UINT_TO_STRING(DATA.BUF_COUNT);
			CASE x OF
			01:	LOG_CL.PRINTF[4] := DATA.D_STRING;
			02:	LOG_CL.PRINTF[4] := REAL_TO_STRING(DATA.D_REAL);
			03:	LOG_CL.PRINTF[4] := DWORD_TO_STRH(DATA.D_DWORD);
			ELSE
				LOG_CL.PRINTF[4] := '';
			END_CASE;
			LOG_MSG();
		END_IF;*)
		(*########################################################################*)
	END_IF;

	IF (mode_last = 10 AND DATA.D_MODE = 11) OR (mode_last = 12 AND DATA.D_MODE = 0) THEN (* löschen nur direkt nach lesen möglich *)
		mode_last := DATA.D_MODE;
		DATA.BUF_SIZE := DATA.BUF_SIZE - cnt - HeaderSize;
		DATA.BUF_COUNT := DATA.BUF_COUNT - 1;
		DATA._First := DATA._GetEnd;
		DATA.BUF_USED := UINT_TO_USINT(100 * DATA.BUF_SIZE / SIZEOF(DATA.BUF)); (* benützer Speicher in % *)
		DATA.D_MODE := 0;

		(*####################  DEBUG-MESSAGE  ###################################*)
		(*IF _debug_enable THEN
			LOG_CL.NEW_MSG := 'RP: DEL /HEAD ~1 / SIZE ~2 / CNT ~3 / >~4<';
			LOG_CL.PRINTF[1] := DWORD_TO_STRH(DATA.D_HEAD);
			LOG_CL.PRINTF[2] := UINT_TO_STRING(cnt);
			LOG_CL.PRINTF[3] := UINT_TO_STRING(DATA.BUF_COUNT);
			CASE x OF
			01:	LOG_CL.PRINTF[4] := DATA.D_STRING;
			02:	LOG_CL.PRINTF[4] := REAL_TO_STRING(DATA.D_REAL);
			03:	LOG_CL.PRINTF[4] := DWORD_TO_STRH(DATA.D_DWORD);
			ELSE
				LOG_CL.PRINTF[4] := '';
			END_CASE;
			LOG_MSG();
		END_IF;*)
		(*########################################################################*)
	END_IF;

99:	(* Buffer reset - alles löschen *)
	DATA._First := 0;
	DATA._Last := 0;
	DATA._GetStart := 0;
	DATA._GetEnd := 0;
	DATA.BUF_COUNT := 0;
	DATA.BUF_SIZE := 0;
	DATA.BUF_USED := 0;
	DATA.D_STRING := '';
	DATA.D_DWORD := 0;
	DATA.D_REAL := 0.0;
	DATA.D_HEAD := 0;
	DATA.D_MODE := 0;
	mode_last := 0;
END_CASE;

(* revision history
ks	01. jan. 2011	rev 1.0
	original version
ks	25. july. 2011	rev 1.1
	neuen MODE 12 hinzugefügt
*)

END_FUNCTION_BLOCK

// oscat_network/POUs/DEMO/BASE64_DEMO_1
PROGRAM BASE64_DEMO_1
VAR
	text1: STRING(144) := '<4036.1076324381@guildenstern.zeitform.de>';
	text2: STRING(192);
	text3: STRING(144);
	BASE64_DECODE_STR: BASE64_DECODE_STR;
	BASE64_ENCODE_STR: BASE64_ENCODE_STR;
	start: BOOL := TRUE;
	done1: BOOL;
	done2: BOOL;
END_VAR

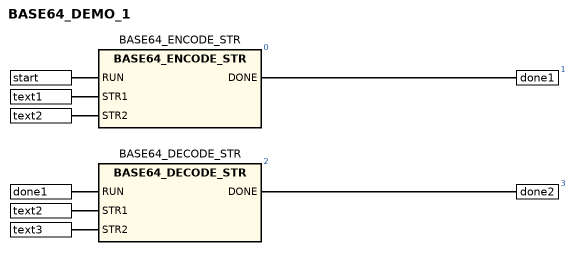
BASE64_ENCODE_STR(RUN := start, STR1 := text1, STR2 := text2);
done1 := BASE64_ENCODE_STR.DONE;
BASE64_DECODE_STR(RUN := done1, STR1 := text2, STR2 := text3);
done2 := BASE64_DECODE_STR.DONE;

END_PROGRAM

// oscat_network/POUs/DEMO/CSV_PARSER_BUF_DEMO_1
PROGRAM CSV_PARSER_BUF_DEMO_1
VAR CONSTANT
	 line_cnt : INT:=2;
	 col_cnt : INT:=4;
END_VAR
VAR
	CPB : CSV_PARSER_BUF;
	FS : FILE_SERVER;
	FSD : FILE_SERVER_DATA;
	PT : NETWORK_BUFFER;
	sep : BYTE;
	value : STRING(STRING_LENGTH);
	step : INT;
	result : BYTE;
	offset : UDINT;
	run : BYTE;
	done : BOOL;
	value_real : REAL;
	cnt : INT;
	line : INT;
	idx : INT;
	data : ARRAY [1..line_cnt, 1..col_cnt] OF REAL;

	(*LOG_MSG : LOG_MSG;
	_debug_enable : BOOL := TRUE;*)
END_VAR

(* Demo-Programm: CSV-Datei mittels Enumeration auswerten
die groesse des arrays kann mittels konstanten line_cnt und col_cnt angepasst werden

 ----- den nachfolgenden Textblock als datei "csv.txt" auf der sps ablegen ---
10.45,20,30,40.8
115,3450.2123,456,123.1
---------------------------------------------------------------------------------*)

CASE step OF

00:	IF NOT done THEN
	 	(* File_Daten einrichten  *)
		FSD.FILENAME := 'csv.txt'; (* Dateiname *)
		FSD.MODE := 1; (* vorhandene Datei zum lesen öffnen *)
		FSD.OFFSET := 0; (* Start bei Dateianfang *)
		FSD.AUTO_CLOSE := T#0s; (* kein Auto-Close verwenden *)
		PT.SIZE := 65535; (* maximale länge einlesen *)
		step := 10;
	END_IF;

10:	IF FSD.MODE = 0 THEN (* Datei geöffnet ? *)
		OFFSET := 0; (* Start Offset vorgeben *)
		sep :=44; (* Trennzeichen , *)
		run := 1; (* Element suchen *)
		cnt := 0;
		step := 20;
	END_IF;

20:	IF run = 0 THEN
		(* ---------------------- Debug-Message ----------------------------*)
		(*IF _debug_enable THEN
			LOG_CL.NEW_MSG := 'CPFD: /value >~2< /offset ~3 /Run ~4 /Result ~5';
			LOG_CL.PRINTF[2] := value;
			LOG_CL.PRINTF[3] := UDINT_TO_STRING(OFFSET);
			LOG_CL.PRINTF[4] := BYTE_TO_STRING(run);
			LOG_CL.PRINTF[5] := BYTE_TO_STRING(result);
			LOG_MSG();
		END_IF;*)
		(* -----------------------------------------------------------------*)

		run := 1; (*  nächstes Element suchen  *)

		IF result = 1 OR result = 2 THEN
			(* automatische konvertierung in real ausführen *)
			IF LEN(value) <= 20 THEN
				value_real := FLOAT_TO_REAL(FLT:=value);
			ELSE
				value_real := 0.0;
			END_IF;

			cnt := cnt + 1;
			IF cnt <= line_cnt * col_cnt THEN
				line := (cnt / col_cnt) + 1;
				idx := (cnt MOD col_cnt);
				data[line,idx] := value_real; (* Daten in Array eintragen *)
			END_IF;

		ELSIF result = 10 THEN (* nichts mehr gefunden *)
			run := 0; (* keine weitere INI Auswertung erwünscht *)
			FSD.MODE := 5; (* Datei schliessen *)
			step := 30;
		END_IF;
	END_IF;

30:	IF FSD.MODE = 0 THEN (* Datei geschlossen ? *)
		step := 0;
		done := TRUE;
	END_IF;

END_CASE;

CPB(SEP:=sep,RUN:=run,OFFSET:=OFFSET,VALUE:=value,PT:=PT,RESULT=>result); (* CSV PARAMETER BUF *)
FS(FSD:=FSD,PT:=PT); (* FILE_SERVER *)

END_PROGRAM

// oscat_network/POUs/DEMO/CSV_PARSER_FILE_DEMO_1
PROGRAM CSV_PARSER_FILE_DEMO_1
VAR CONSTANT
	 line_cnt : INT:=2;
	 col_cnt : INT:=4;
END_VAR
VAR
	CPF : CSV_PARSER_FILE;
	FS : FILE_SERVER;
	FSD : FILE_SERVER_DATA;
	PT : NETWORK_BUFFER;
	filename : STRING;
	value :	STRING(STRING_LENGTH);
	sep : BYTE;
	step : INT;
	result : BYTE;
	offset : UDINT;
	run : BYTE;
	done : BOOL;
	value_real : REAL;
	cnt : INT;
	line : INT;
	idx : INT;
	data : ARRAY [1..line_cnt, 1..col_cnt] OF REAL;

	(*LOG_MSG : LOG_MSG;
	_debug_enable : BOOL := TRUE;*)
END_VAR

(* Demo-Programm: CSV-Datei mittels Enumeration auswerten

die groesse des arrays kann mittels konstanten line_cnt und col_cnt angepasst werden

 ----- den nachfolgenden Textblock als datei "csv.txt" auf der sps ablegen ---
10.45,20,30,40.8
115,3450.2123,456,123.1
---------------------------------------------------------------------------------*)

CASE step OF

00:	IF NOT done THEN
		filename := 'csv.txt'; (* File_Daten einrichten *)
		OFFSET := 0; (* Start Offset vorgeben *)
		FSD.AUTO_CLOSE := T#0ms; (* kein Automatisches schliessen *)
		sep :=44; (* Trennzeichen , *)
		run := 1; (* Element suchen *)
		cnt := 0;
		step := 20;
	END_IF;

20:	IF run = 0 THEN (* kein Befehl mehr aktiv ? *)
		(* ---------------------- Debug-Message ----------------------------*)
		(*IF _debug_enable THEN
			LOG_CL.NEW_MSG := 'CPFD: /value >~2< /offset ~3 /Run ~4 /Result ~5';
			LOG_CL.PRINTF[2] := value;
			LOG_CL.PRINTF[3] := UDINT_TO_STRING(OFFSET);
			LOG_CL.PRINTF[4] := BYTE_TO_STRING(run);
			LOG_CL.PRINTF[5] := BYTE_TO_STRING(result);
			LOG_MSG();
		END_IF;*)
		(* -----------------------------------------------------------------*)

		run := 1; (*  nächstes Element suchen  *)

		IF result = 1 OR result = 2 THEN
			(* automatische konvertierung in real ausführen *)
			IF LEN(value) <= 20 THEN
				value_real := FLOAT_TO_REAL(FLT:=value);
			ELSE
				value_real := 0.0;
			END_IF;

			cnt := cnt + 1;
			IF cnt <= line_cnt * col_cnt THEN
				line := (cnt / col_cnt) + 1;
				idx := (cnt MOD col_cnt);
				data[line,idx] := value_real; (* Daten in Array eintragen *)
			END_IF;

		ELSIF result = 10 THEN (* nichts mehr gefunden *)
			run := 0; (* keine weitere INI Auswertung erwünscht *)
			FSD.MODE := 5; (* Datei schliessen *)
			step := 30;
		END_IF;
	END_IF;

30:	IF FSD.MODE = 0 THEN (* Befehl Datei schliessen beendet *)
		step := 0;
		done := TRUE;
	END_IF;

END_CASE;

CPF(SEP:=sep,FILENAME:=FILENAME,FSD:=FSD,RUN:=run,OFFSET:=OFFSET,VALUE:=value,PT:=PT,RESULT=>result); (* CSV PARAMETER FILE *)
FS(FSD:=FSD,PT:=PT); (* FILE_SERVER *)

END_PROGRAM

// oscat_network/POUs/DEMO/DLOG_FILE_CSV_DEMO_1
PROGRAM DLOG_FILE_CSV_DEMO_1
VAR
	RTC_2: RTC_2;
	x : DLOG_DATA;
	DLOG_STORE_FILE_CSV : DLOG_STORE_FILE_CSV;
	CLK_PRG: CLK_PRG;
	cur_dt: DT;
	enable: BOOL;
	rtc_set : BOOL := TRUE;

	trig_t : UDINT := 0;
	trig_m : BOOL;

	x1: DLOG_DT;
	x2 : DLOG_REAL;
	x3 : DLOG_DINT;
	x4 : DLOG_BOOL;
	x5: DLOG_STRING;
	GEN_SIN_1: GEN_SIN;
	COUNT_DR: COUNT_DR;
	error_c: DWORD;
	error_t: BYTE;
END_VAR

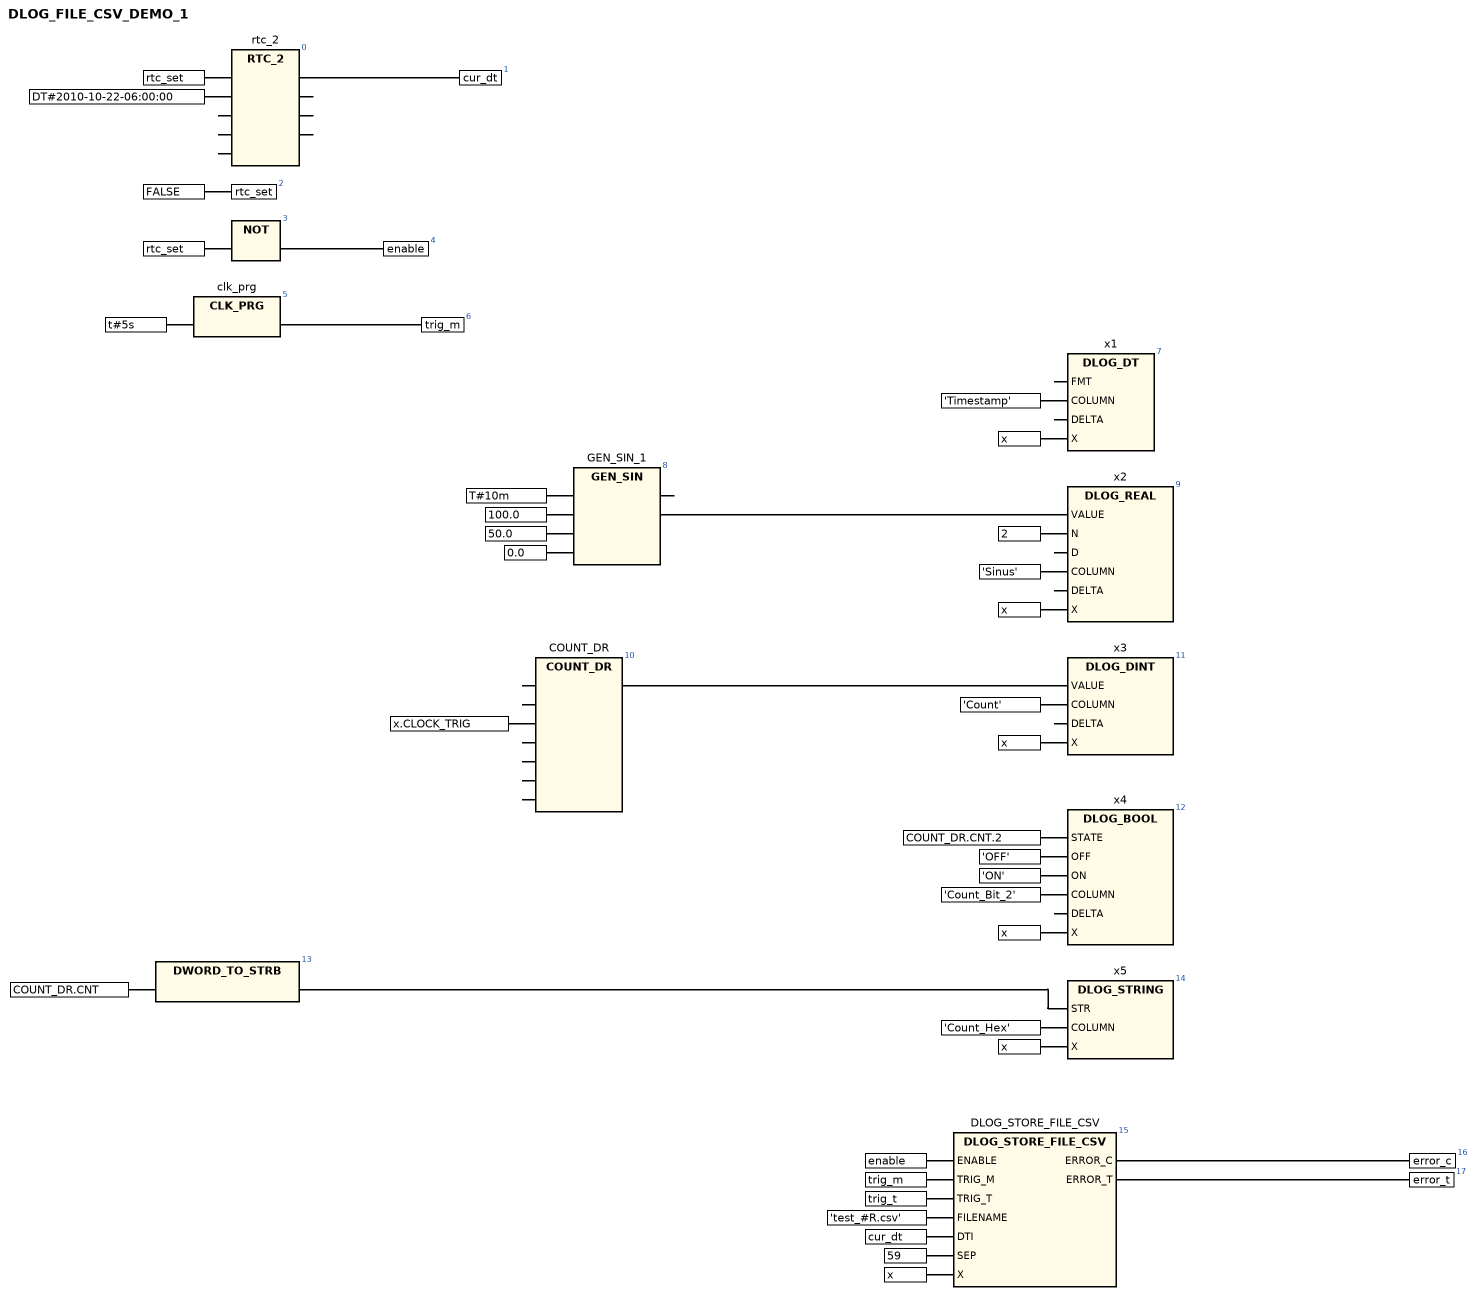
rtc_2(_in1 := rtc_set, _in2 := DT#2010-10-22-06:00:00);
cur_dt := rtc_2._out1;
rtc_set := FALSE;
enable := NOT rtc_set;
clk_prg(_in1 := t#5s);
trig_m := clk_prg._out1;
x1(COLUMN := 'Timestamp', X := x); // DLOG_DT
GEN_SIN_1(_in1 := T#10m, _in2 := 100.0, _in3 := 50.0, _in4 := 0.0); // GEN_SIN
x2(VALUE := GEN_SIN_1._out2, N := 2, COLUMN := 'Sinus', X := x); // DLOG_REAL
COUNT_DR(_in3 := x.CLOCK_TRIG);
x3(VALUE := COUNT_DR._out1, COLUMN := 'Count', X := x); // DLOG_DINT
x4(STATE := COUNT_DR.CNT.2, OFF := 'OFF', ON := 'ON', COLUMN := 'Count_Bit_2', X := x); // DLOG_BOOL
x5(STR := DWORD_TO_STRB(COUNT_DR.CNT), COLUMN := 'Count_Hex', X := x); // DLOG_STRING
DLOG_STORE_FILE_CSV(
    ENABLE := enable,
    TRIG_M := trig_m,
    TRIG_T := trig_t,
    FILENAME := 'test_#R.csv',
    DTI := cur_dt,
    SEP := 59,
    X := x);
error_c := DLOG_STORE_FILE_CSV.ERROR_C;
error_t := DLOG_STORE_FILE_CSV.ERROR_T;

END_PROGRAM

// oscat_network/POUs/DEMO/DLOG_FILE_CSV_FTP_DEMO_1
PROGRAM DLOG_FILE_CSV_FTP_DEMO_1
VAR
	RTC_2: RTC_2;
	x : DLOG_DATA;
	DLOG_STORE_FILE_CSV : DLOG_STORE_FILE_CSV;
	CLK_PRG: CLK_PRG;
	cur_dt: DT;
	enable: BOOL;
	rtc_set : BOOL := TRUE;

	trig_t : UDINT := 0;
	trig_m : BOOL;

	x1: DLOG_DT;
	x2 : DLOG_REAL;
	x3 : DLOG_DINT;
	x4 : DLOG_BOOL;
	x5: DLOG_STRING;
	GEN_SIN_1: GEN_SIN;
	COUNT_DR: COUNT_DR;
	error_c: DWORD;
	error_t: BYTE;

	DLOG_FILE_TO_FTP: DLOG_FILE_TO_FTP;
	ftp_done: BOOL;
	ftp_busy: BOOL;
	ftp_error_c: DWORD;
	ftp_error_t: BYTE;
	ftp_url: STRING := 'ftp://581920:123456@oscat.atwebpages.com:2000/subordner/';
	ftp_activ: BOOL := FALSE;
	ftp_delete: BOOL := TRUE;
	ftp_retry: INT := 0;
	ftp_retry_time: TIME := T#60s;
	ftp_timeout: TIME := T#30s;
END_VAR
VAR // added by the converter: edge detectors and wires of the graphical bodies
    _w1, _w2 : ANY;
END_VAR

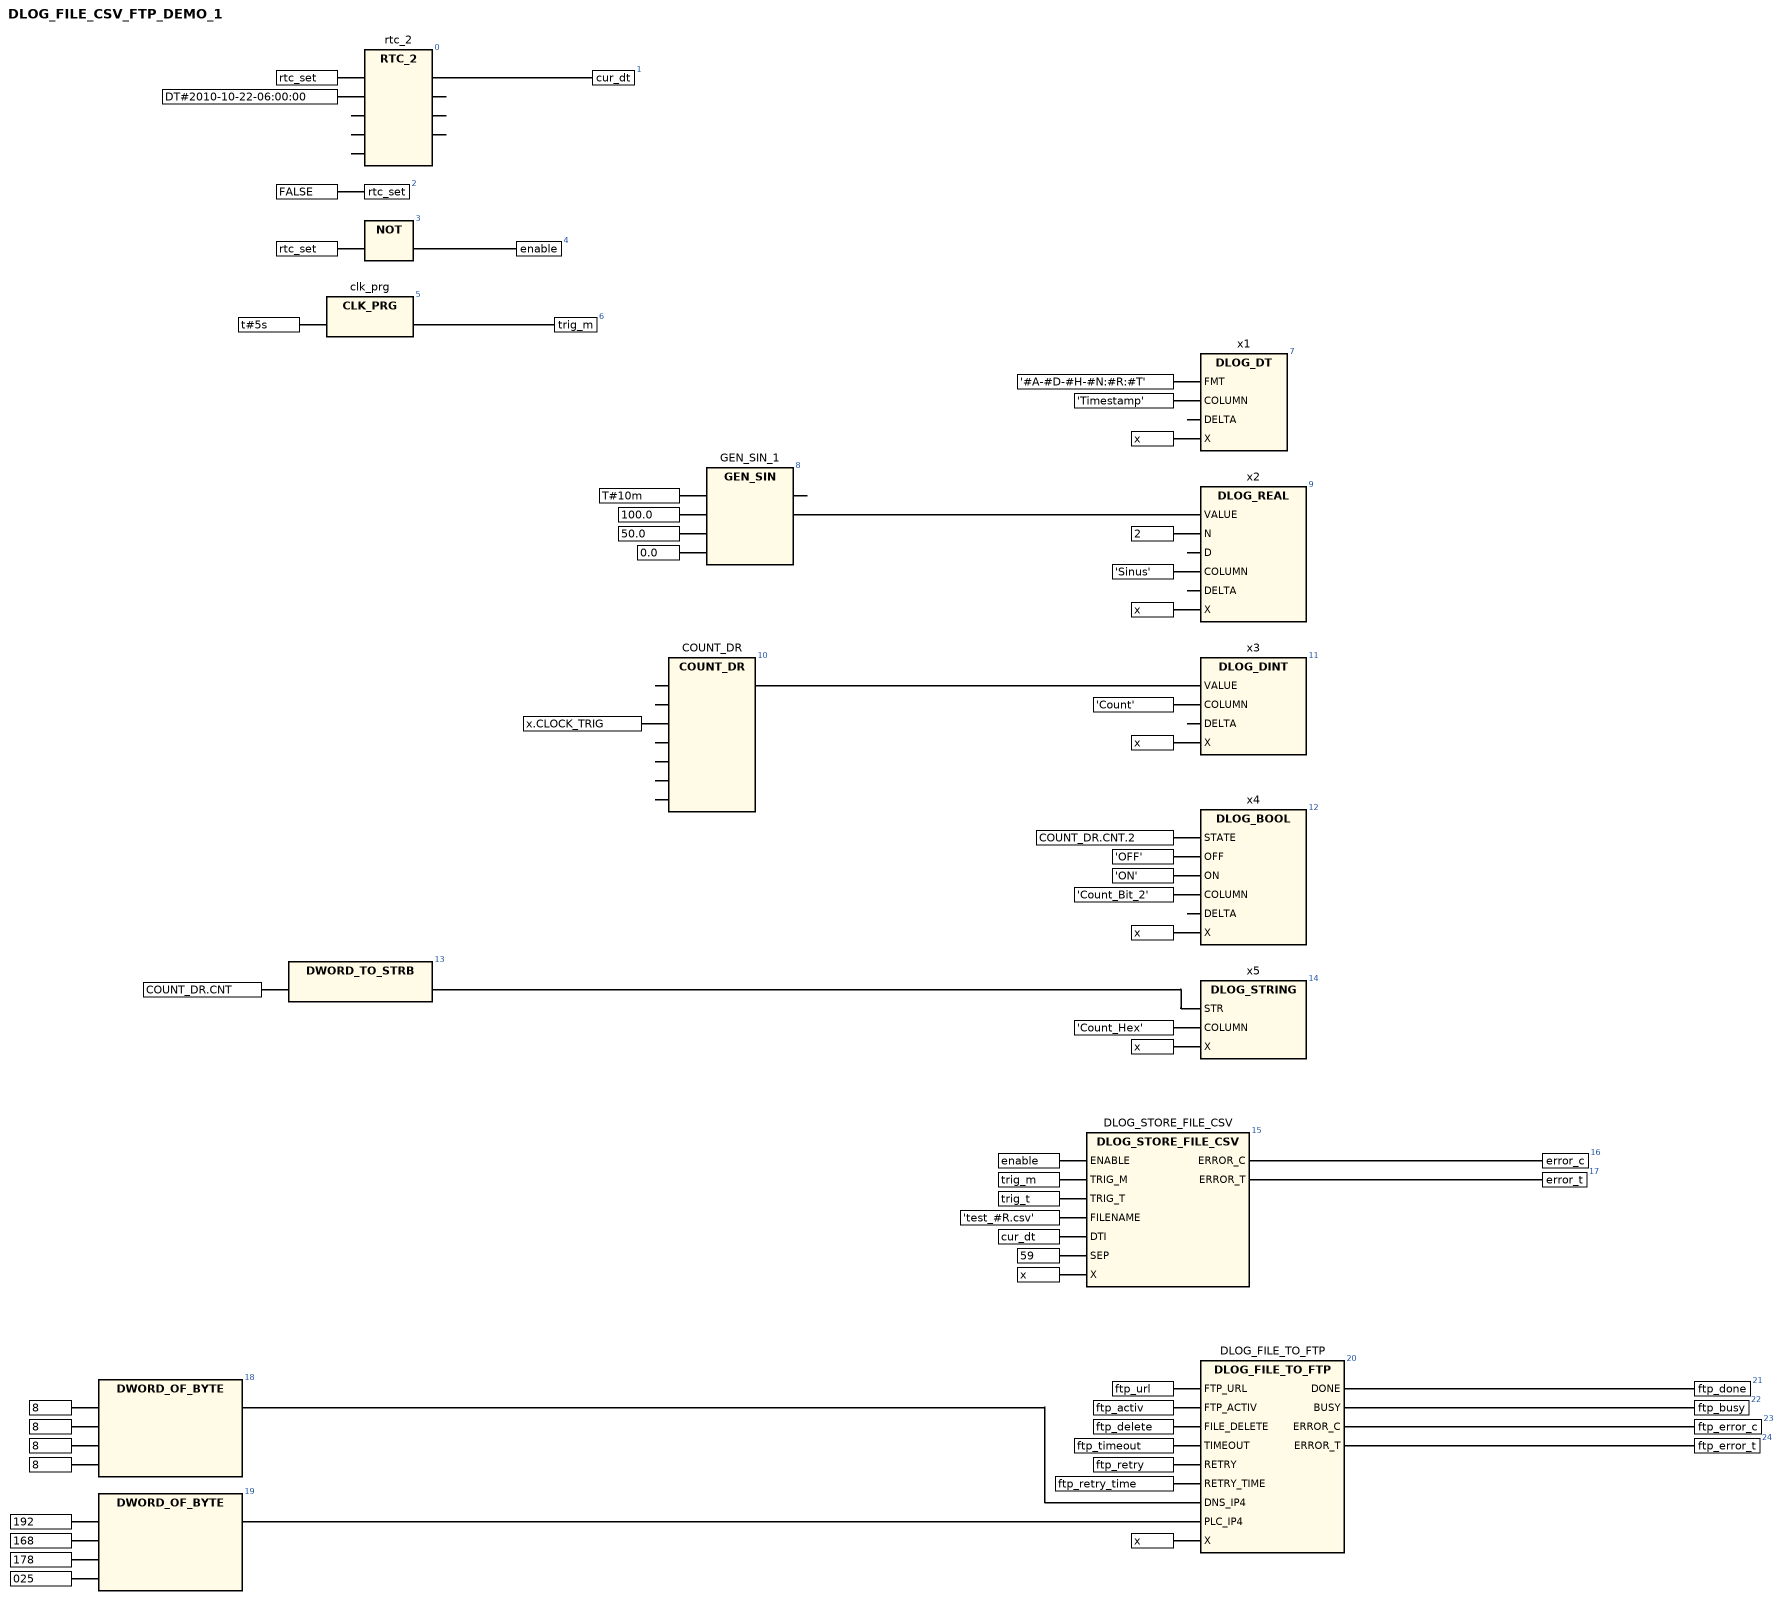
rtc_2(_in1 := rtc_set, _in2 := DT#2010-10-22-06:00:00);
cur_dt := rtc_2._out1;
rtc_set := FALSE;
enable := NOT rtc_set;
clk_prg(_in1 := t#5s);
trig_m := clk_prg._out1;
x1(FMT := '#A-#D-#H-#N:#R:#T', COLUMN := 'Timestamp', X := x); // DLOG_DT
GEN_SIN_1(_in1 := T#10m, _in2 := 100.0, _in3 := 50.0, _in4 := 0.0); // GEN_SIN
x2(VALUE := GEN_SIN_1._out2, N := 2, COLUMN := 'Sinus', X := x); // DLOG_REAL
COUNT_DR(_in3 := x.CLOCK_TRIG);
x3(VALUE := COUNT_DR._out1, COLUMN := 'Count', X := x); // DLOG_DINT
x4(STATE := COUNT_DR.CNT.2, OFF := 'OFF', ON := 'ON', COLUMN := 'Count_Bit_2', X := x); // DLOG_BOOL
x5(STR := DWORD_TO_STRB(COUNT_DR.CNT), COLUMN := 'Count_Hex', X := x); // DLOG_STRING
DLOG_STORE_FILE_CSV(
    ENABLE := enable,
    TRIG_M := trig_m,
    TRIG_T := trig_t,
    FILENAME := 'test_#R.csv',
    DTI := cur_dt,
    SEP := 59,
    X := x);
error_c := DLOG_STORE_FILE_CSV.ERROR_C;
error_t := DLOG_STORE_FILE_CSV.ERROR_T;
_w1 := DWORD_OF_BYTE(8, 8, 8, 8);
_w2 := DWORD_OF_BYTE(192, 168, 178, 025);
DLOG_FILE_TO_FTP(
    FTP_URL := ftp_url,
    FTP_ACTIV := ftp_activ,
    FILE_DELETE := ftp_delete,
    TIMEOUT := ftp_timeout,
    RETRY := ftp_retry,
    RETRY_TIME := ftp_retry_time,
    DNS_IP4 := _w1,
    PLC_IP4 := _w2,
    X := x);
ftp_done := DLOG_FILE_TO_FTP.DONE;
ftp_busy := DLOG_FILE_TO_FTP.BUSY;
ftp_error_c := DLOG_FILE_TO_FTP.ERROR_C;
ftp_error_t := DLOG_FILE_TO_FTP.ERROR_T;

END_PROGRAM

// oscat_network/POUs/DEMO/DLOG_FILE_CSV_SMTP_DEMO_1
PROGRAM DLOG_FILE_CSV_SMTP_DEMO_1
VAR
	RTC_2: RTC_2;
	x : DLOG_DATA;
	DLOG_STORE_FILE_CSV : DLOG_STORE_FILE_CSV;
	CLK_PRG: CLK_PRG;
	cur_dt: DT;
	enable: BOOL;
	rtc_set : BOOL := TRUE;

	trig_t : UDINT := 0;
	trig_m : BOOL;

	x1: DLOG_DT;
	x2 : DLOG_REAL;
	x3 : DLOG_DINT;
	x4 : DLOG_BOOL;
	x5: DLOG_STRING;
	GEN_SIN_1: GEN_SIN;
	COUNT_DR: COUNT_DR;
	error_c: DWORD;
	error_t: BYTE;

	DLOG_FILE_TO_SMTP: DLOG_FILE_TO_SMTP;
	smtp_timeout: TIME := T#30s;
	smtp_error_t: BYTE;
	smtp_error_c: DWORD;
	smtp_busy: BOOL;
	smtp_done: BOOL;
	smtp_dti: DT;
	smtp_dti_offset: INT := 60;
	smtp_server: STRING := '110876022:oscat123456@mail.gmx.net';
	smtp_mailfrom: STRING := 'oscat@gmx.net;Station_01';
	smtp_mailto: STRING(STRING_LENGTH) := 'oscat@gmx.net';
	smtp_subject: STRING := 'Das ist der Betreff';
	smtp_body: STRING(STRING_LENGTH) := 'Das ist der Email-Text';
	smtp_delete: BOOL := TRUE;
	smtp_retry: INT := 0;
	smtp_retry_time: TIME := T#60s;
END_VAR
VAR // added by the converter: edge detectors and wires of the graphical bodies
    _w1 : ANY;
END_VAR

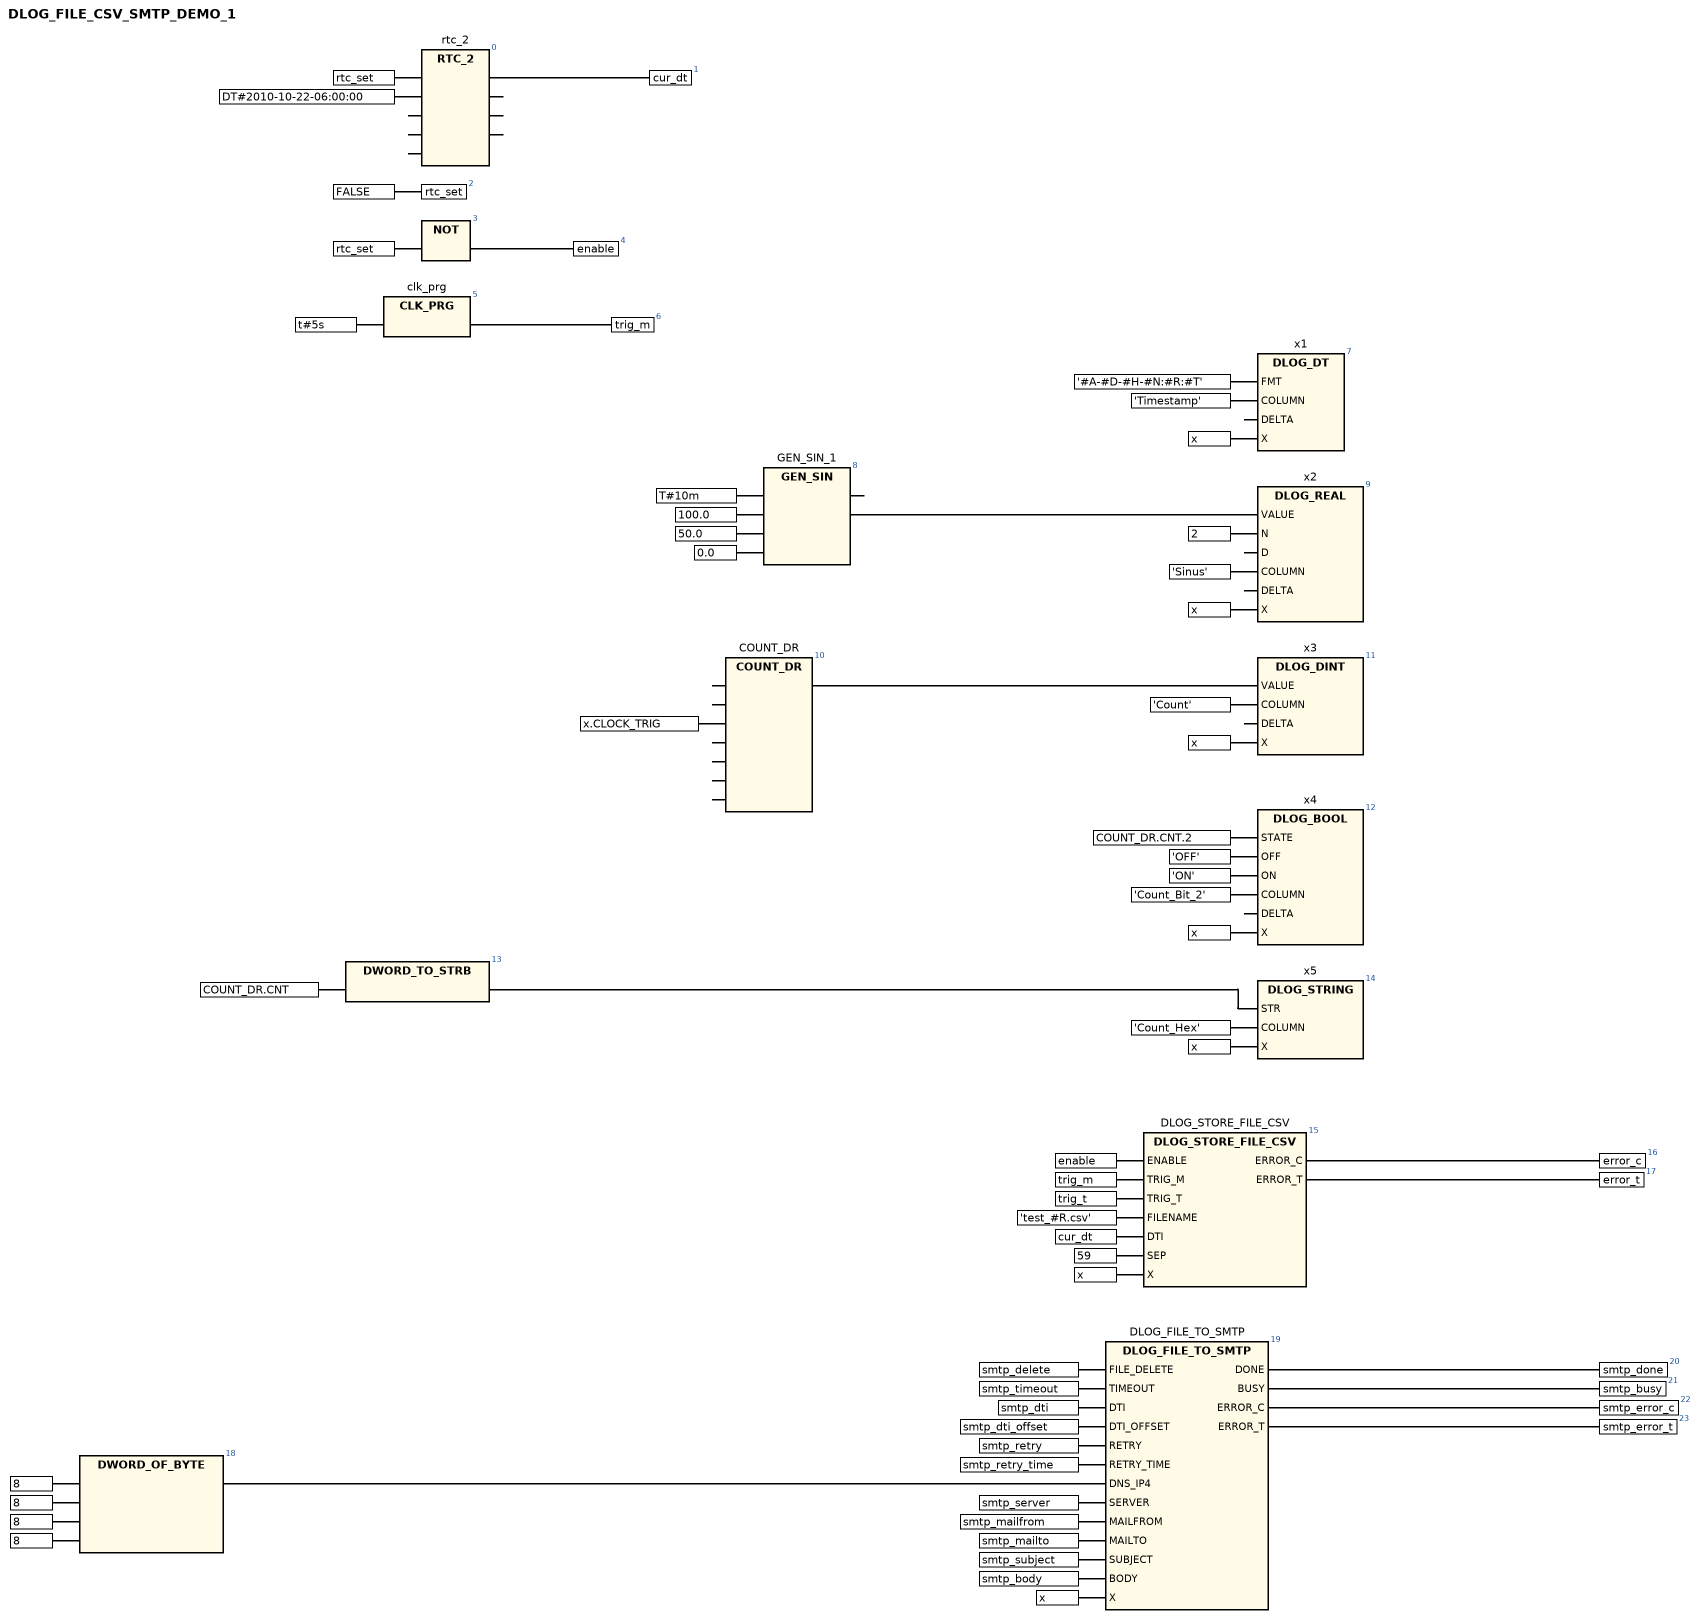
rtc_2(_in1 := rtc_set, _in2 := DT#2010-10-22-06:00:00);
cur_dt := rtc_2._out1;
rtc_set := FALSE;
enable := NOT rtc_set;
clk_prg(_in1 := t#5s);
trig_m := clk_prg._out1;
x1(FMT := '#A-#D-#H-#N:#R:#T', COLUMN := 'Timestamp', X := x); // DLOG_DT
GEN_SIN_1(_in1 := T#10m, _in2 := 100.0, _in3 := 50.0, _in4 := 0.0); // GEN_SIN
x2(VALUE := GEN_SIN_1._out2, N := 2, COLUMN := 'Sinus', X := x); // DLOG_REAL
COUNT_DR(_in3 := x.CLOCK_TRIG);
x3(VALUE := COUNT_DR._out1, COLUMN := 'Count', X := x); // DLOG_DINT
x4(STATE := COUNT_DR.CNT.2, OFF := 'OFF', ON := 'ON', COLUMN := 'Count_Bit_2', X := x); // DLOG_BOOL
x5(STR := DWORD_TO_STRB(COUNT_DR.CNT), COLUMN := 'Count_Hex', X := x); // DLOG_STRING
DLOG_STORE_FILE_CSV(
    ENABLE := enable,
    TRIG_M := trig_m,
    TRIG_T := trig_t,
    FILENAME := 'test_#R.csv',
    DTI := cur_dt,
    SEP := 59,
    X := x);
error_c := DLOG_STORE_FILE_CSV.ERROR_C;
error_t := DLOG_STORE_FILE_CSV.ERROR_T;
_w1 := DWORD_OF_BYTE(8, 8, 8, 8);
DLOG_FILE_TO_SMTP(
    FILE_DELETE := smtp_delete,
    TIMEOUT := smtp_timeout,
    DTI := smtp_dti,
    DTI_OFFSET := smtp_dti_offset,
    RETRY := smtp_retry,
    RETRY_TIME := smtp_retry_time,
    DNS_IP4 := _w1,
    SERVER := smtp_server,
    MAILFROM := smtp_mailfrom,
    MAILTO := smtp_mailto,
    SUBJECT := smtp_subject,
    BODY := smtp_body,
    X := x);
smtp_done := DLOG_FILE_TO_SMTP.DONE;
smtp_busy := DLOG_FILE_TO_SMTP.BUSY;
smtp_error_c := DLOG_FILE_TO_SMTP.ERROR_C;
smtp_error_t := DLOG_FILE_TO_SMTP.ERROR_T;

END_PROGRAM

// oscat_network/POUs/DEMO/DLOG_FILE_HTML_DEMO_1
PROGRAM DLOG_FILE_HTML_DEMO_1
VAR
	RTC_2: RTC_2;
	x : DLOG_DATA;
	DLOG_STORE_FILE_HTML: DLOG_STORE_FILE_HTML;
	CLK_PRG: CLK_PRG;
	cur_dt: DT;
	enable: BOOL := TRUE;
	rtc_set : BOOL := TRUE;

	trig_t : UDINT := 0;
	trig_m : BOOL;

	x1: DLOG_DT;
	x2 : DLOG_REAL;
	x3 : DLOG_DINT;
	x4 : DLOG_BOOL;
	x5: DLOG_STRING;
	GEN_SIN_1: GEN_SIN;
	COUNT_DR: COUNT_DR;
	error_c: DWORD;
	error_t: BYTE;

	html_caption: STRING := 'Das ist der Titel';
	html_tr_even: STRING := 'BGCOLOR=#B3B7FF';
	html_tr_odd: STRING := 'BGCOLOR=#E0E0E0';
	html_tr_head: STRING := 'BGCOLOR=#FFFF40';
	html_table : STRING := 'BORDER="1"';
END_VAR

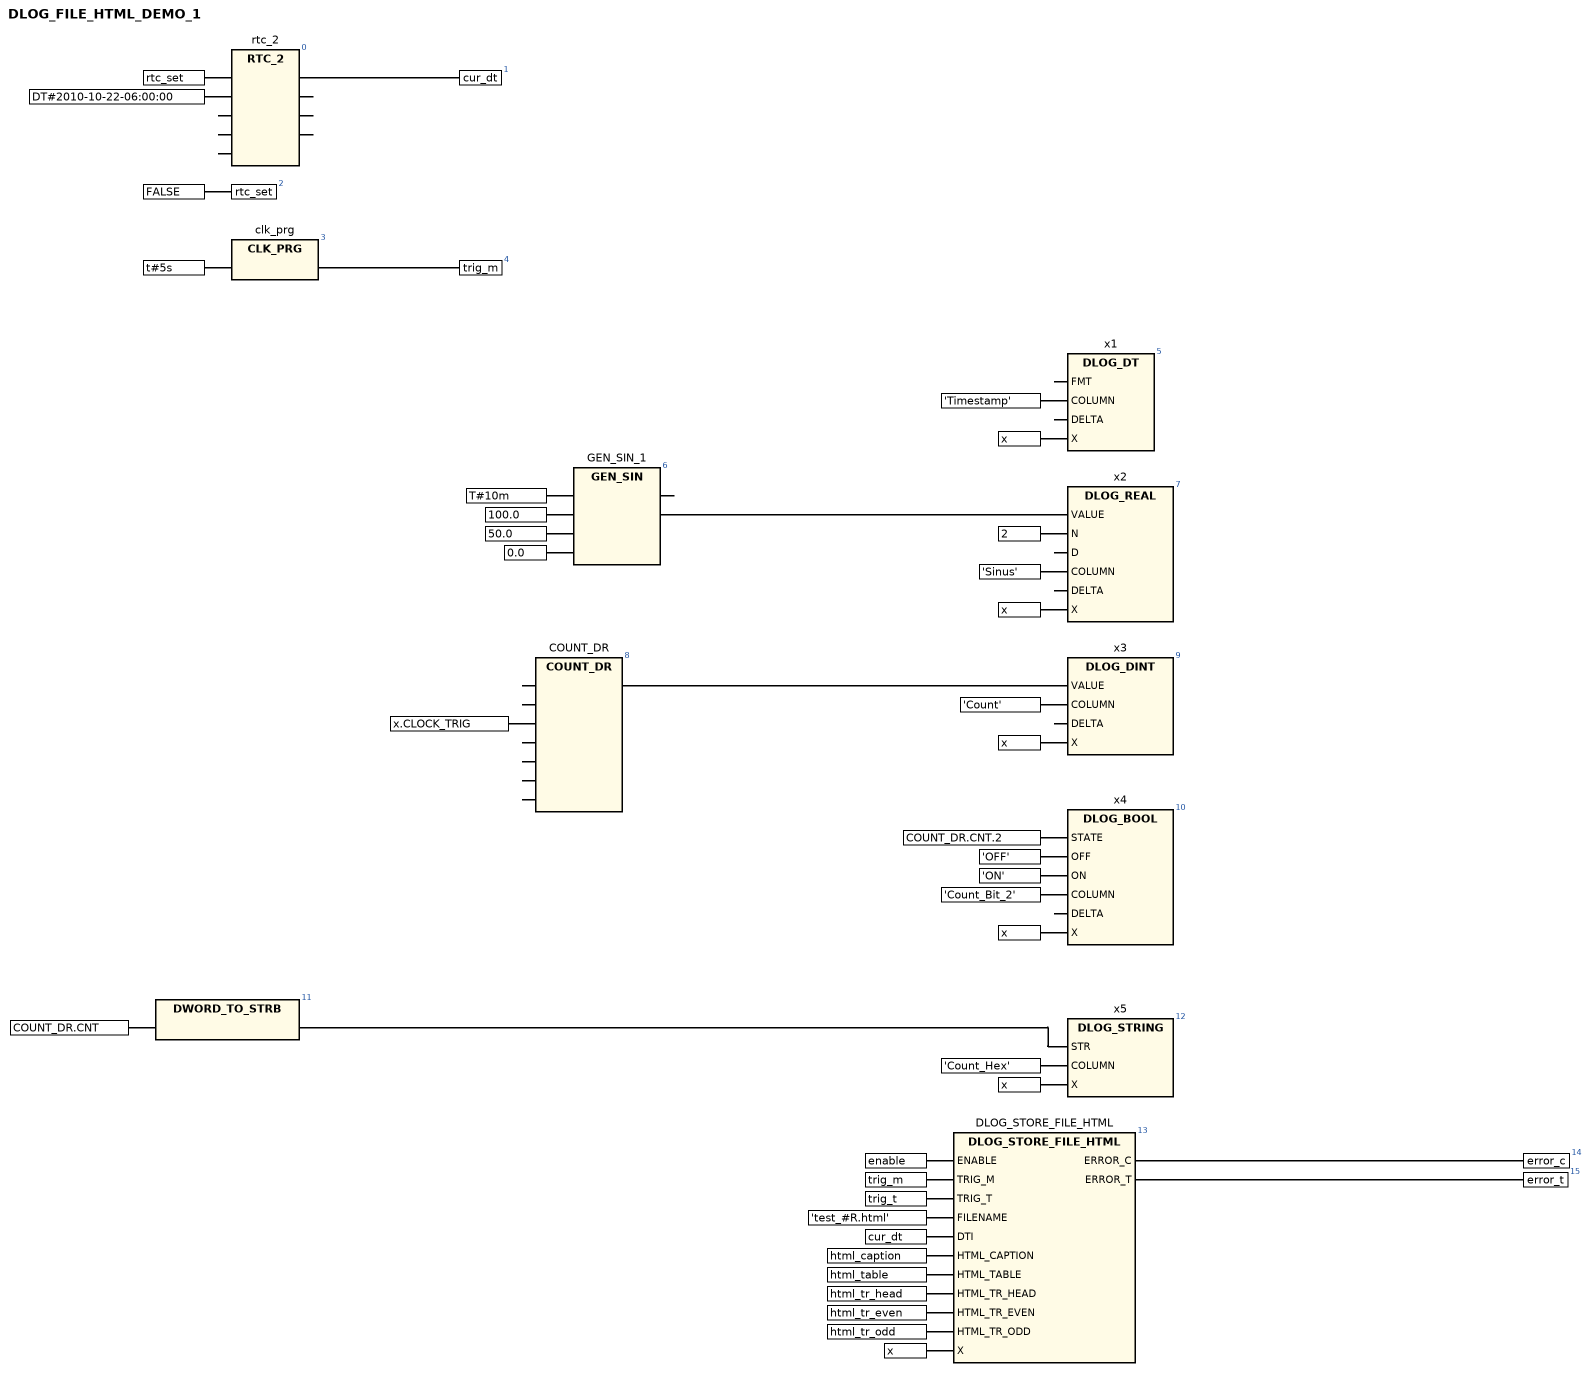
rtc_2(_in1 := rtc_set, _in2 := DT#2010-10-22-06:00:00);
cur_dt := rtc_2._out1;
rtc_set := FALSE;
clk_prg(_in1 := t#5s);
trig_m := clk_prg._out1;
x1(COLUMN := 'Timestamp', X := x); // DLOG_DT
GEN_SIN_1(_in1 := T#10m, _in2 := 100.0, _in3 := 50.0, _in4 := 0.0); // GEN_SIN
x2(VALUE := GEN_SIN_1._out2, N := 2, COLUMN := 'Sinus', X := x); // DLOG_REAL
COUNT_DR(_in3 := x.CLOCK_TRIG);
x3(VALUE := COUNT_DR._out1, COLUMN := 'Count', X := x); // DLOG_DINT
x4(STATE := COUNT_DR.CNT.2, OFF := 'OFF', ON := 'ON', COLUMN := 'Count_Bit_2', X := x); // DLOG_BOOL
x5(STR := DWORD_TO_STRB(COUNT_DR.CNT), COLUMN := 'Count_Hex', X := x); // DLOG_STRING
DLOG_STORE_FILE_HTML(
    ENABLE := enable,
    TRIG_M := trig_m,
    TRIG_T := trig_t,
    FILENAME := 'test_#R.html',
    DTI := cur_dt,
    HTML_CAPTION := html_caption,
    HTML_TABLE := html_table,
    HTML_TR_HEAD := html_tr_head,
    HTML_TR_EVEN := html_tr_even,
    HTML_TR_ODD := html_tr_odd,
    X := x);
error_c := DLOG_STORE_FILE_HTML.ERROR_C;
error_t := DLOG_STORE_FILE_HTML.ERROR_T;

END_PROGRAM

// oscat_network/POUs/DEMO/DLOG_FILE_XML_DEMO_1
PROGRAM DLOG_FILE_XML_DEMO_1
VAR
	RTC_2: RTC_2;
	x : DLOG_DATA;
	DLOG_STORE_FILE_XML: DLOG_STORE_FILE_XML;
	CLK_PRG: CLK_PRG;
	cur_dt: DT;
	enable: BOOL := TRUE;
	rtc_set : BOOL := TRUE;

	trig_t : UDINT := 0;
	trig_m : BOOL;

	x1: DLOG_DT;
	x2 : DLOG_REAL;
	x3 : DLOG_DINT;
	x4 : DLOG_BOOL;
	x5: DLOG_STRING;
	GEN_SIN_1: GEN_SIN;
	COUNT_DR: COUNT_DR;
	error_c: DWORD;
	error_t: BYTE;
END_VAR

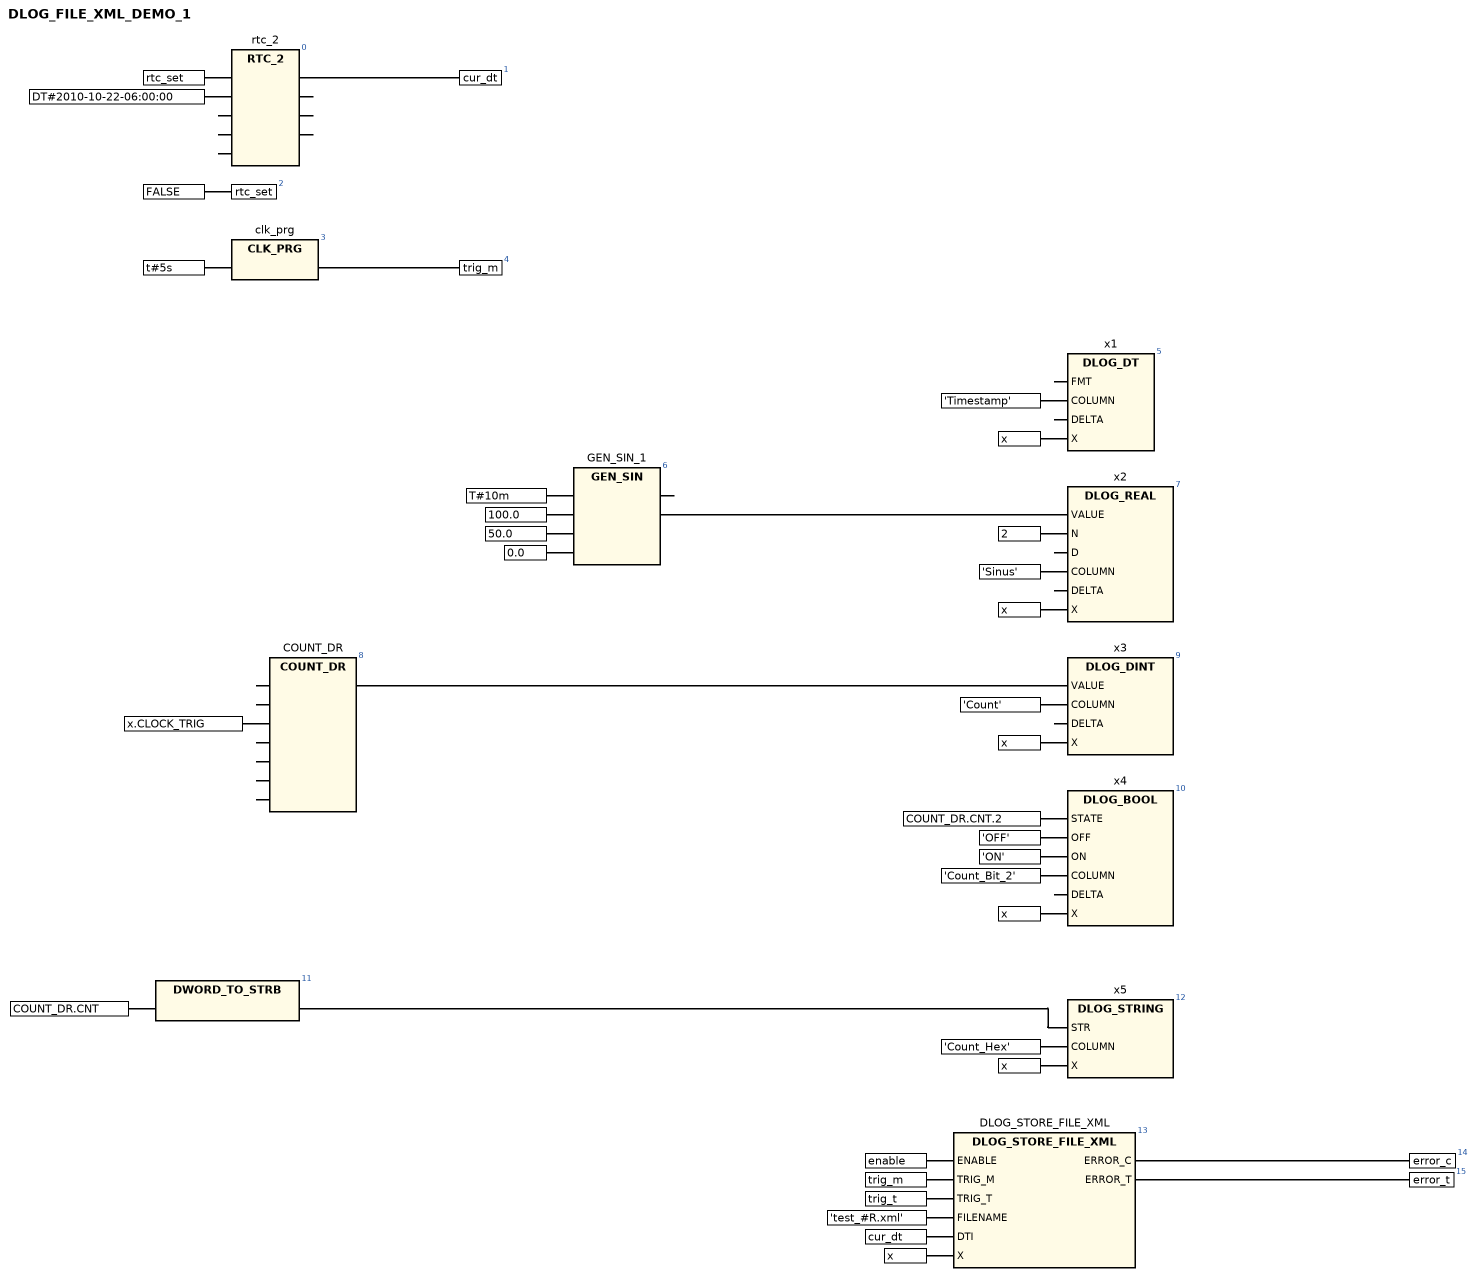
rtc_2(_in1 := rtc_set, _in2 := DT#2010-10-22-06:00:00);
cur_dt := rtc_2._out1;
rtc_set := FALSE;
clk_prg(_in1 := t#5s);
trig_m := clk_prg._out1;
x1(COLUMN := 'Timestamp', X := x); // DLOG_DT
GEN_SIN_1(_in1 := T#10m, _in2 := 100.0, _in3 := 50.0, _in4 := 0.0); // GEN_SIN
x2(VALUE := GEN_SIN_1._out2, N := 2, COLUMN := 'Sinus', X := x); // DLOG_REAL
COUNT_DR(_in3 := x.CLOCK_TRIG);
x3(VALUE := COUNT_DR._out1, COLUMN := 'Count', X := x); // DLOG_DINT
x4(STATE := COUNT_DR.CNT.2, OFF := 'OFF', ON := 'ON', COLUMN := 'Count_Bit_2', X := x); // DLOG_BOOL
x5(STR := DWORD_TO_STRB(COUNT_DR.CNT), COLUMN := 'Count_Hex', X := x); // DLOG_STRING
DLOG_STORE_FILE_XML(
    ENABLE := enable,
    TRIG_M := trig_m,
    TRIG_T := trig_t,
    FILENAME := 'test_#R.xml',
    DTI := cur_dt,
    X := x);
error_c := DLOG_STORE_FILE_XML.ERROR_C;
error_t := DLOG_STORE_FILE_XML.ERROR_T;

END_PROGRAM

// oscat_network/POUs/DEMO/DLOG_RRD_DEMO_1
PROGRAM DLOG_RRD_DEMO_1
VAR
	RTC_2 : RTC_2;
	CLK_PRG: CLK_PRG;
	cur_dt : DT;
	rtc_set : BOOL := TRUE;
	enable : BOOL := TRUE;
	DLOG_STORE_RRD : DLOG_STORE_RRD;
	trig_t : UDINT := 0;
	trig_m : BOOL;

	rrd_error_c : DWORD;
	rrd_error_t : BYTE;
	rrd_enable : BOOL := TRUE;
	rrd_url : STRING(STRING_LENGTH) := 'http://xxx.com/myhouse/rrd/test_rrd.php?rrd_db=test.rrd&value=';
	rrd_timeout: TIME := t#5s;

	x : DLOG_DATA;
	x1 : DLOG_DINT;
	x2 : DLOG_DINT;
	x3 : DLOG_REAL;
	x4 : DLOG_REAL;
	x5 : DLOG_REAL;
	x6 : DLOG_REAL;
	x7 : DLOG_REAL;

	GEN_SIN_1 : GEN_SIN;
	GEN_SIN_2 : GEN_SIN;
	GEN_SIN_3 : GEN_SIN;
	GEN_RMP_1: GEN_RMP;
	GEN_RMP_2: GEN_RMP;
END_VAR
VAR // added by the converter: edge detectors and wires of the graphical bodies
    _w1, _w2, _w3 : ANY;
END_VAR

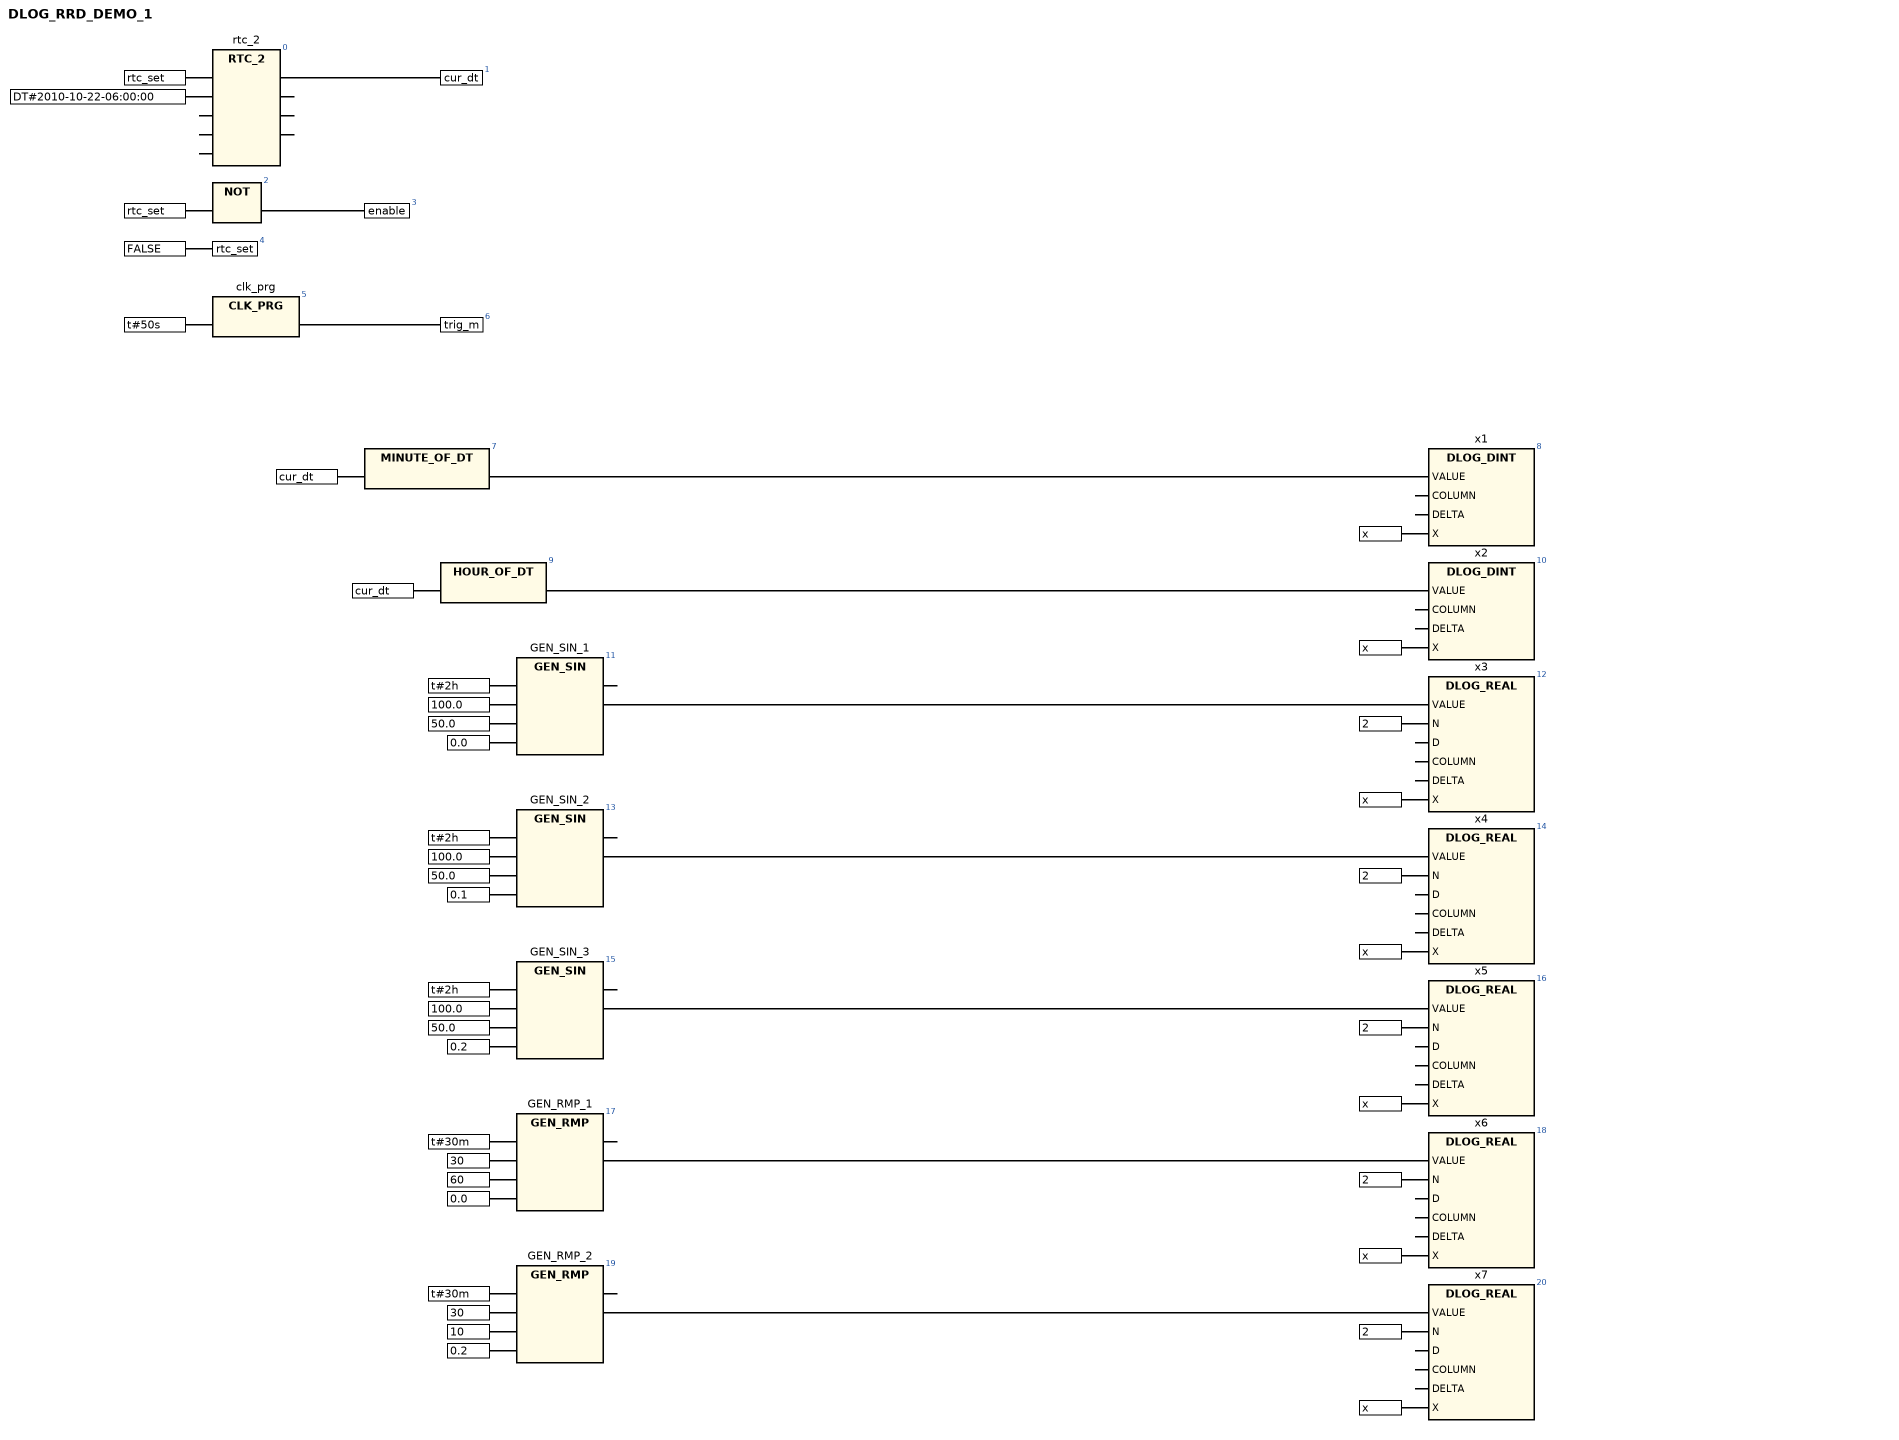
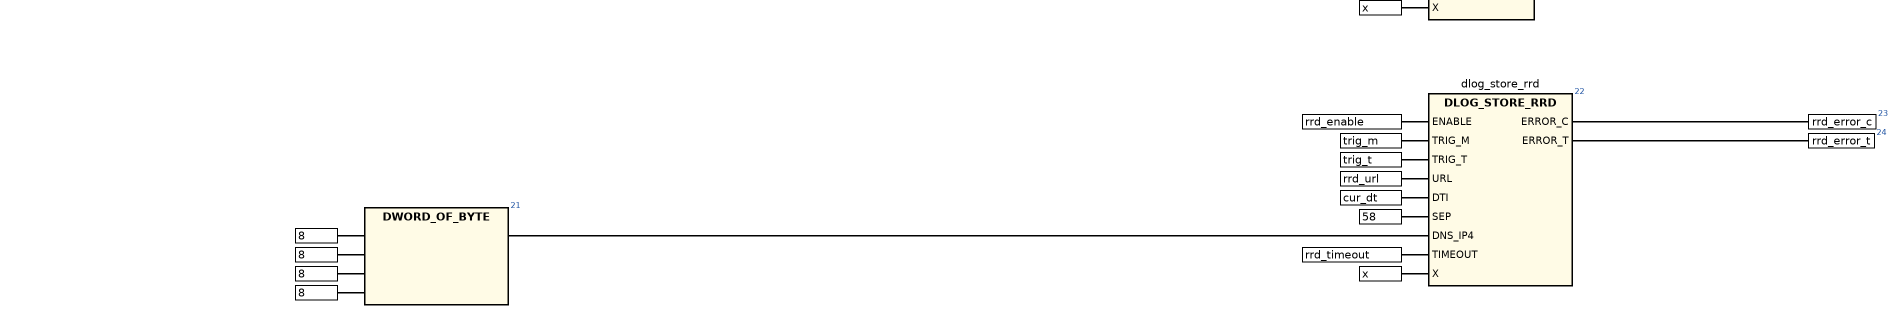
rtc_2(_in1 := rtc_set, _in2 := DT#2010-10-22-06:00:00);
cur_dt := rtc_2._out1;
enable := NOT rtc_set;
rtc_set := FALSE;
clk_prg(_in1 := t#50s);
trig_m := clk_prg._out1;
_w1 := MINUTE_OF_DT(cur_dt);
x1(VALUE := _w1, X := x); // DLOG_DINT
_w2 := HOUR_OF_DT(cur_dt);
x2(VALUE := _w2, X := x); // DLOG_DINT
GEN_SIN_1(_in1 := t#2h, _in2 := 100.0, _in3 := 50.0, _in4 := 0.0); // GEN_SIN
x3(VALUE := GEN_SIN_1._out2, N := 2, X := x); // DLOG_REAL
GEN_SIN_2(_in1 := t#2h, _in2 := 100.0, _in3 := 50.0, _in4 := 0.1); // GEN_SIN
x4(VALUE := GEN_SIN_2._out2, N := 2, X := x); // DLOG_REAL
GEN_SIN_3(_in1 := t#2h, _in2 := 100.0, _in3 := 50.0, _in4 := 0.2); // GEN_SIN
x5(VALUE := GEN_SIN_3._out2, N := 2, X := x); // DLOG_REAL
GEN_RMP_1(_in1 := t#30m, _in2 := 30, _in3 := 60, _in4 := 0.0); // GEN_RMP
x6(VALUE := GEN_RMP_1._out2, N := 2, X := x); // DLOG_REAL
GEN_RMP_2(_in1 := t#30m, _in2 := 30, _in3 := 10, _in4 := 0.2); // GEN_RMP
x7(VALUE := GEN_RMP_2._out2, N := 2, X := x); // DLOG_REAL
_w3 := DWORD_OF_BYTE(8, 8, 8, 8);
dlog_store_rrd(
    ENABLE := rrd_enable,
    TRIG_M := trig_m,
    TRIG_T := trig_t,
    URL := rrd_url,
    DTI := cur_dt,
    SEP := 58,
    DNS_IP4 := _w3,
    TIMEOUT := rrd_timeout,
    X := x);
rrd_error_c := dlog_store_rrd.ERROR_C;
rrd_error_t := dlog_store_rrd.ERROR_T;

END_PROGRAM

// oscat_network/POUs/DEMO/DNS_DYN_DEMO_1
PROGRAM DNS_DYN_DEMO_1
VAR
	DNS_DYN : DNS_DYN;
	IP_C : IP_C;
	S_BUF : NETWORK_BUFFER;
	R_BUF : NETWORK_BUFFER;
	IP_CONTROL : IP_CONTROL;
	enable: BOOL;
	done : BOOL;
	error_c : DWORD;
	error_t : BYTE;
	busy : BOOL;
	COUNT_DR: COUNT_DR;
	z: DWORD;

	GET_WAN_IP : GET_WAN_IP;
	t1: TON;
	done2 : BOOL;
	error_c2 : DWORD;
	error_t2 : BYTE;
	update : BOOL;
	new_ip: BOOL;
	wan_ip4: DWORD;
END_VAR
VAR // added by the converter: edge detectors and wires of the graphical bodies
    _w1 : ANY;
END_VAR

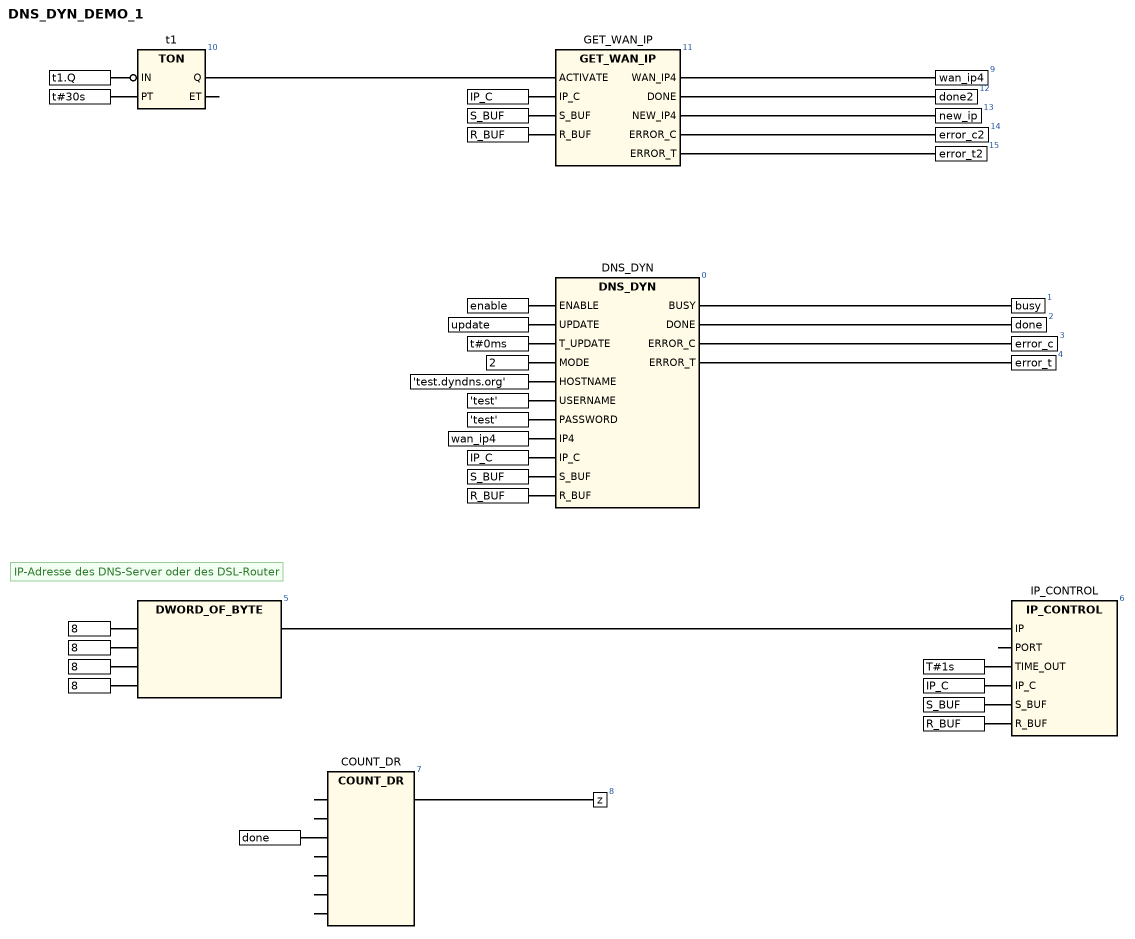
DNS_DYN(
    ENABLE := enable,
    UPDATE := update,
    T_UPDATE := t#0ms,
    MODE := 2,
    HOSTNAME := 'test.dyndns.org',
    USERNAME := 'test',
    PASSWORD := 'test',
    IP4 := wan_ip4,
    IP_C := IP_C,
    S_BUF := S_BUF,
    R_BUF := R_BUF);
busy := DNS_DYN.BUSY;
done := DNS_DYN.DONE;
error_c := DNS_DYN.ERROR_C;
error_t := DNS_DYN.ERROR_T;
// IP-Adresse des DNS-Server oder des DSL-Router
_w1 := DWORD_OF_BYTE(8, 8, 8, 8);
IP_CONTROL(IP := _w1, TIME_OUT := T#1s, IP_C := IP_C, S_BUF := S_BUF, R_BUF := R_BUF);
COUNT_DR(_in3 := done);
z := COUNT_DR._out1;
wan_ip4 := GET_WAN_IP.WAN_IP4;
t1(IN := NOT t1.Q, PT := t#30s); // TON
GET_WAN_IP(ACTIVATE := t1.Q, IP_C := IP_C, S_BUF := S_BUF, R_BUF := R_BUF);
done2 := GET_WAN_IP.DONE;
new_ip := GET_WAN_IP.NEW_IP4;
error_c2 := GET_WAN_IP.ERROR_C;
error_t2 := GET_WAN_IP.ERROR_T;

END_PROGRAM

// oscat_network/POUs/NETWORK/DNS_DYN
FUNCTION_BLOCK DNS_DYN
VAR_IN_OUT
	IP_C : IP_C; (* IP_Control Verwaltungsstruktur *)
	S_BUF : NETWORK_BUFFER;
	R_BUF : NETWORK_BUFFER;
END_VAR
VAR_INPUT
	ENABLE : BOOL;
	UPDATE : BOOL;
	T_UPDATE : TIME := T#1h;
	MODE : BYTE;
	HOSTNAME : STRING(30);
	USERNAME : STRING(20);
	PASSWORD : STRING(20);
	IP4 : DWORD;
END_VAR
VAR_OUTPUT
	BUSY : BOOL;
	DONE : BOOL;
	ERROR_C : DWORD;
	ERROR_T : BYTE;
END_VAR
VAR
	DNS_CLIENT : DNS_CLIENT;
	HTTP_GET : HTTP_GET;
	BASE64_ENCODE_STR : BASE64_ENCODE_STR;
	URL_DATA : url;
	update_last : BOOL;
	state : INT;
	base64_done : BOOL;
	s1 : STRING(144);
	s2 : STRING(192);
	w : TON;
END_VAR

(*

version 1.2		02. dec. 2009
programmer 		ks
tested by		ks

YAHOO_WEATHER lädt vom Yahoo-Webserver einen Wetter RSS-Feed und analysiert die Daten und legt diese in einem Array ab
*)

CASE state OF

00:	IF ENABLE AND ((UPDATE AND NOT update_last) OR w.Q) THEN
		state := 20;
		DONE := FALSE;
		BUSY := TRUE;
		ERROR_C := DWORD#0;
		ERROR_T := BYTE#0;

		IF MODE = 0 THEN (* dyndns.org *)
			s2 := CONCAT('http://members.dyndns.org/nic/update?hostname=',HOSTNAME);
		ELSE (* selfhost.de *)
			s2 := 'http://carol.selfhost.de/nic/update?hostname=1';
		END_IF;
		IF IP4 > 0 THEN (* parametrierte IP verwenden *)
			s1 := CONCAT('&myip=',IP4_TO_STRING(IP4));
			s2 := CONCAT(s2,s1);
		END_IF;
		URL_DATA:=STRING_TO_URL(STR:=s2, DEFAULT_PROTOCOL:='', DEFAULT_PATH:=''); (* URL for DNS UND HTTP-GET *)
		s1 := CONCAT(USERNAME,':');
		s1 := CONCAT(s1,PASSWORD); (* BASE64 Encode Text *)
	END_IF;

20:	IF DNS_CLIENT.DONE THEN (* DNS_CLIENT *)
			state := 40;
	ELSIF (DNS_CLIENT.ERROR > DWORD#00) THEN (* Fehlerbehandlung *)
		ERROR_C := DNS_CLIENT.ERROR;
		ERROR_T := BYTE#01;
		BUSY := FALSE;
		state := 0;
	END_IF;

40: IF base64_done THEN (* BASE64 Encode beendet ? *)
		s1 := CONCAT('Authorization: Basic ',s2);
		s1 := CONCAT(s1,'$0D$0AUser-Agent: x$0D$0A');
		URL_DATA.HEADER := s1;
		state := 60;
	END_IF;

60:	IF HTTP_GET.DONE THEN
		state := 0;
		BUSY := FALSE;
		DONE := TRUE;

		(* !! Codes !!
		Successful Updates: 		good , nchg
		Update Syntax Errors:		badsys , badagent
		Account-Related Errors:		badauth , !donator
		Hostname-Related Errors:	notfqdn , nohost , !yours , numhost , abuse
		Server Error Conditions:	dnserr , 911
		*)
		s2 := BUFFER_TO_STRING(PT:=ADR(R_BUF.BUFFER),SIZE:=SIZEOF(R_BUF.BUFFER),START:=HTTP_GET.BODY_START + 3,STOP:=HTTP_GET.BODY_STOP - 7);
		IF FIND(s2,'good') = 0 THEN
			IF FIND(s2,'nochg') = 0 THEN
				ERROR_C := DWORD#1;
				ERROR_T := BYTE#03;
				DONE := FALSE;
			END_IF;
		END_IF;
	ELSIF (HTTP_GET.ERROR > DWORD#00) THEN (* Fehlerbehandlung *)
		ERROR_C := HTTP_GET.ERROR;
		ERROR_T := BYTE#02;
		BUSY := FALSE;
		state := 0;
	END_IF;

END_CASE;

DNS_CLIENT(IP_C:=IP_C,	S_BUF:=S_BUF, R_BUF:=R_BUF,DOMAIN:=URL_DATA.DOMAIN, IP4_DNS:=0, ACTIVATE:=state=20); (* DNS_CLIENT *)
HTTP_GET( IP_C:=IP_C, S_BUF:=S_BUF, R_BUF:=R_BUF, IP4:=DNS_CLIENT.IP4, GET:=state=60, MODE:=2, UNLOCK_BUF:=state<>60,URL_DATA:=URL_DATA); (* HTTP_GET *)
BASE64_ENCODE_STR( RUN:=state=40, STR1:=s1, STR2:=s2, DONE=>base64_done); (* BASE64 Encode *)

IF T_UPDATE > T#0ms THEN w(IN:=state=0, PT:=T_UPDATE); END_IF;
update_last := UPDATE;

(* revision history
ks	01. jan. 2010	rev 1.0
	original version

*)

END_FUNCTION_BLOCK

// oscat_network/POUs/WEATHER/YAHOO_WEATHER
FUNCTION_BLOCK YAHOO_WEATHER
VAR_IN_OUT
	IP_C : IP_C; (* IP_Control Verwaltungsstruktur *)
	S_BUF : NETWORK_BUFFER;
	R_BUF : NETWORK_BUFFER;
	YW : YAHOO_WEATHER_DATA;
END_VAR
VAR_INPUT
	ACTIVATE : BOOL;
	UNITS : BOOL;
	LOCATION : STRING(20);
END_VAR
VAR_OUTPUT
	BUSY : BOOL;
	DONE : BOOL;
	ERROR_C : DWORD;
	ERROR_T : BYTE;
END_VAR
VAR
	CTRL : XML_CONTROL;
	XML_READER : XML_READER;
	URL_DATA : url;
	DNS_CLIENT : DNS_CLIENT;
	HTTP_GET : HTTP_GET;
	last_state : BOOL;
	value_int : INT;
	value_real : REAL;
	v_real : REAL;
	state : INT;
END_VAR

(*

version 1.3		04. may. 2011
programmer 		ks
tested by			ks

YAHOO_WEATHER lädt vom Yahoo-Webserver einen Wetter RSS-Feed und analysiert die Daten und legt diese in einem Array ab
*)

CASE state OF

00:	IF ACTIVATE AND NOT last_state THEN
		state := 20;
		DONE := FALSE;
		BUSY := TRUE;
		ERROR_C := DWORD#0;
		ERROR_T := BYTE#0;
	END_IF;

20: (* URL for DNS UND HTTP-GET *)
	(* Example: http://weather.yahooapis.com/forecastrss?p=94089&u=c *)
	URL_DATA:=STRING_TO_URL(STR:='http://weather.yahooapis.com/forecastrss',
							DEFAULT_PROTOCOL:='',
							DEFAULT_PATH:=''
							);
  	URL_DATA.QUERY := CONCAT('w=',LOCATION);

	IF UNITS THEN
		URL_DATA.QUERY := CONCAT(URL_DATA.QUERY,'&u=f'); (* fahrenheit *)
	ELSE
		URL_DATA.QUERY := CONCAT(URL_DATA.QUERY,'&u=c'); (* celsius *)
	END_IF;
	state := 40;

40:	IF DNS_CLIENT.DONE THEN
		state := 60;
	ELSIF (DNS_CLIENT.ERROR > DWORD#00) THEN
		(* Fehlerbehandlung *)
		ERROR_C := DNS_CLIENT.ERROR;
	ERROR_T := BYTE#01;
		state   := 100;
	END_IF;

60:	IF HTTP_GET.DONE THEN
		state := 80;
		CTRL.START_POS := HTTP_GET.BODY_START;
		CTRL.STOP_POS := HTTP_GET.BODY_STOP;
		CTRL.COMMAND := WORD#2#10000000_00011000; (* ONLY TEXT AND ATTRIBUTE *)
		CTRL.WATCHDOG  := T#1ms;

	ELSIF (HTTP_GET.ERROR > DWORD#00) THEN
		(* Fehlerbehandlung *)
		ERROR_C := HTTP_GET.ERROR;
		ERROR_T := BYTE#02;
		state := 100;
	END_IF;

80: XML_READER(CTRL:=CTRL,BUF:=R_BUF.BUFFER); (* XML Daten seriell lesen *)
	IF CTRL.TYP < 98 THEN (* nur auswerten wenn kein Watchdog durchlauf *)
		value_int := 0;
		value_real := 0.0;
		(* automatische konvertierung in real und int ausführen *)
		IF LEN(CTRL.VALUE) <= 20 THEN
			v_real:=FLOAT_TO_REAL(FLT:=CTRL.VALUE);
			IF CHK_REAL(v_real) = 0 THEN (* !!! prüft auf gültigen REAL Wert, ansonsten stürzt Twincat ab !!!!  *)
				value_real := v_real;
				value_int := REAL_TO_INT(value_real);
			END_IF;
		END_IF;

		IF CTRL.COUNT < UINT#52 THEN (* Performance-Teilung *)
			(* ------------ Teil 1 --------------*)
			CASE UINT_TO_INT(CTRL.COUNT) OF
			027: YW.TimeToLive := value_int;
			030: YW.location_city := CTRL.VALUE;
			031: YW.location_region := CTRL.VALUE;
			032: YW.location_country := CTRL.VALUE;
			035: YW.unit_temperature := CTRL.VALUE;
			036: YW.unit_distance := CTRL.VALUE;
			037: YW.unit_pressure := CTRL.VALUE;
			038: YW.unit_speed := CTRL.VALUE;
			041: YW.wind_chill := value_int;
			042: YW.wind_direction := value_int;
			043: YW.wind_speed := value_real;
			046: YW.atmosphere_humidity := value_int;
			047: YW.atmosphere_visibility := value_real;
			048: YW.atmosphere_pressure := value_int;
			049: YW.atmosphere_rising := value_int;
			END_CASE;
		ELSE
			(* ------------ Teil 2 --------------*)
			CASE UINT_TO_INT(CTRL.COUNT) OF
			052: YW.astronomy_sunrise := CTRL.VALUE;
			053: YW.astronomy_sunset := CTRL.VALUE;
			077: YW.geo_latitude := value_real;
			080: YW.geo_longitude := value_real;
			089: YW.cur_conditions_text := CTRL.VALUE;
			090: YW.cur_conditions_code := value_int;
				YW.cur_conditions_icon := value_int;
			091: YW.cur_conditions_temp := value_int;
			100: YW.forcast_today_low_temp := value_int;
			101: YW.forcast_today_high_temp := value_int;
			102: YW.forcast_today_text := CTRL.VALUE;
			103: YW.forcast_today_code := value_int;
				YW.forcast_today_icon := value_int;
			108: YW.forcast_tomorrow_low_temp := value_int;
			109: YW.forcast_tomorrow_high_temp := value_int;
			110: YW.forcast_tomorrow_text := CTRL.VALUE;
			111: YW.forcast_tomorrow_code := value_int;
				YW.forcast_tomorrow_icon := value_int;
			END_CASE;
		END_IF;
	ELSIF CTRL.TYP = 99 THEN (* EXIT - letztes Element gelesen *)
		DONE  := TRUE;
		state := 100;
	END_IF; 

100:
	(* UNLOCK HTTP DATA *)
	IF (NOT HTTP_GET.DONE) THEN
		state := 0;
		BUSY := FALSE;
		DONE := ERROR_T = BYTE#0;
	END_IF; 

	END_CASE;

(* ---------------- DNS --------------- *)
DNS_CLIENT(	IP_C:=IP_C,
			S_BUF:=S_BUF,
			R_BUF:=R_BUF,
			DOMAIN:=URL_DATA.DOMAIN,
			IP4_DNS:=DWORD#00,
			ACTIVATE:=state=40 (* DNS Start *)
			);
(* nicht oder nicht direkt verwendete Parameter *)
(*	DWORD :=DNS_CLIENT.IP4;
	BOOL  :=DNS_CLIENT.DONE;
	BYTE  :=DNS_CLIENT.ERROR; *)
(* -------------------------------------*)

(* ------------- HTTP_GET --------------- *)
HTTP_GET(	IP_C:=IP_C,
			S_BUF:=S_BUF,
			R_BUF:=R_BUF,
			IP4:=DNS_CLIENT.IP4,
			GET:=state=60,
			MODE:=BYTE#2, (* HTTP 1.1 mit persistenter Verbindung *)
			UNLOCK_BUF:=state=100,
			URL_DATA:=URL_DATA
			);

(* nicht oder nicht direkt verwendete Parameter *)
(*	STRING := HTTP_GET.HTTP_STATUS;
	UINT :=HTTP_GET.HEADER_START;
	UINT :=HTTP_GET.HEADER_STOP;
	UINT :=HTTP_GET.BODY_START;
	UINT :=HTTP_GET.BODY_STOP;
	BOOL :=HTTP_GET.DONE;
	BYTE :=HTTP_GET.ERROR;
*)
(* -------------------------------------*)

last_state := ACTIVATE;

(* revision history
ks	18. dez. 2008	rev 1.0
	original version

ks	01. oct. 2009	rev 1.1
	YAHOO_WEATHER_DATA

ks	24. sep. 2010	rev 1.2
	new URL-Location-parameter and REAL_CHECK (TwinCat BUG) 

ks	04. may. 2011	rev 1.3
	neue elemente:  CUR_CONDITIONS_ICON, FORCAST_TODAY_ICON, FORCAST_TOMORROW_ICON

*)

END_FUNCTION_BLOCK

// oscat_network/POUs/NETWORK/XML_READER
FUNCTION_BLOCK XML_READER
VAR_IN_OUT
	CTRL : XML_CONTROL;
	BUF : NW_BUF_LONG;
END_VAR
VAR
	index :	INT;
	index2 : INT;
	stop : INT;
	mode : INT;
	command : WORD;
	c :	BYTE;
	s1 : INT;
	e1 : INT;
	path_overflow : BOOL;
	empty_tag : BOOL;
	s_code : STRING(10);
	e_code : STRING(10);
	watchdog : TON;

	(*LOG_MSG : LOG_MSG;
	_debug_enable : BOOL := TRUE;*)

END_VAR

(*

version 1.2		10. mai 2010
programmer 	ks
tested by		ks

XML_READER ermöglicht das serielle Parsen und die Auswertung von XML_Elementen in einem Buffer
*)

(*

TYP
00 = UNBEKANNT
01 = ELEMENT (STANDARD)
02 = CLOSE ELEMENT 
03 = TEXT
04 = ATTRIBUTE
05 = ELEMENT (PROCESSING INSTRUCTION) 

12 = !CDATA
13 = !COMMENT
14 = !DTD ELEMENT (Document Type Declarations )

98 = WATCHDOG
99 = ENDE

Bei Typ 02 werden keine Blockdaten ausgegeben !

*)

(* ---------- Init -------------- *)
IF BIT_OF_DWORD(WORD_TO_DWORD(CTRL.COMMAND),15) THEN
	COMMAND := CTRL.COMMAND;
	CTRL.COMMAND := WORD#0;

	index := UINT_TO_INT(CTRL.START_POS);
	stop := UINT_TO_INT(CTRL.STOP_POS);
	mode := 100;
	path_overflow := FALSE;

	CTRL.TYP := 0;
	CTRL.COUNT := UINT#00;
	CTRL.LEVEL := UINT#00;
	CTRL.ATTRIBUTE := '';
	CTRL.ELEMENT := '';
	CTRL.PATH := '';
	CTRL.VALUE := '';

	WATCHDOG.PT := CTRL.WATCHDOG;
END_IF;

(*----------------------------------------------- *)

IF index < 0 THEN RETURN;END_IF;

CTRL.BLOCK1_START := UINT#0;
CTRL.BLOCK1_STOP := UINT#0;
CTRL.BLOCK2_START := UINT#0;
CTRL.BLOCK2_STOP := UINT#0;

WATCHDOG(IN:=FALSE); (* Timer stoppen *)

WHILE (TRUE) DO

